# B&R Automation Studio project NAEUL004C00R13L518F00 (part 21)

#### Act_OptP0935UpdtDat.st
```iecst
ACTION Act_OptP0935UpdtDat:

	tyP0935Lifter.tyMotionStd.tyNumCurrPos.diValue			:= p_diLifterBtmActualPos;
	tyP0935Lifter.tyMotionStd.tyNumErrCode.diValue			:= UDINT_TO_DINT(p_udiLifterBtmAxisErrID);
	tyP0935Lifter.tyMotionStd.tyBitmapPwr.usiValueIdx		:= BOOL_TO_USINT(p_bLifterBtmPwrOn);
	tyP0935Lifter.tyMotionStd.tyBitmapRst.usiValueIdx		:= BOOL_TO_USINT(NOT p_bLifterBtmAxisErr);
	tyP0935Lifter.tyMotionStd.tyBitmapOrigin.usiValueIdx	:= BOOL_TO_USINT(p_bLifterBtmIsHomed);
	tyP0935Lifter.tyMotionStd.tyBtnUpLmtSen.bValue			:= p_bLifterBtmUpSen;
	tyP0935Lifter.tyMotionStd.tyBtnDownLmtSen.bValue		:= p_bLifterBtmDownSen;

	//Machine Bitmap
	IF p_bLifterBtmIsHomed = TRUE THEN
		IF p_diLifterBtmActualPos <= (p_tyNtParamCurr.tyUILifterTargetPos.diMax / 3) THEN
			tyP0935Lifter.tyMotionStd.tyBitmapMc.uiValueIdx 	:= 2;
		ELSIF p_diLifterBtmActualPos <= (p_tyNtParamCurr.tyUILifterTargetPos.diMax / 3 * 2) THEN
			tyP0935Lifter.tyMotionStd.tyBitmapMc.uiValueIdx 	:= 3;
		ELSE
			tyP0935Lifter.tyMotionStd.tyBitmapMc.uiValueIdx 	:= 4;
		END_IF
	ELSE
		tyP0935Lifter.tyMotionStd.tyBitmapMc.uiValueIdx	:= 2;
	END_IF

//	IF p_tyNtParamCurr.eProjMag = ULMagTriple THEN
//		tyP0935Lifter.tyMotionStd.tyBitmapMc.uiValueIdx	:= tyP0935Lifter.tyMotionStd.tyBitmapMc.uiValueIdx + 100;
//	END_IF

	IF p_tyNtParamCurr.eProjMag = ULMagDual THEN
		IF p_tyNtParamCurr.bProjLifterMagPlatform AND p_tyNtParamCurr.bUIConvDirRL THEN
			IF 	tyP0935Lifter.tyMotionStd.tyBitmapMc.uiValueIdx < 700 THEN
				tyP0935Lifter.tyMotionStd.tyBitmapMc.uiValueIdx	:= tyP0935Lifter.tyMotionStd.tyBitmapMc.uiValueIdx + 700;
			END_IF
		ELSIF p_tyNtParamCurr.bProjLifterMagPlatform THEN
			IF p_tyNtParamCurr.bProjMagConvLane1Prep = FALSE THEN
				IF 	tyP0935Lifter.tyMotionStd.tyBitmapMc.uiValueIdx < 600 THEN
					tyP0935Lifter.tyMotionStd.tyBitmapMc.uiValueIdx	:= tyP0935Lifter.tyMotionStd.tyBitmapMc.uiValueIdx + 600;
				END_IF
			ELSE
				IF 	tyP0935Lifter.tyMotionStd.tyBitmapMc.uiValueIdx < 900 THEN //Lifter1 - 902,903,904
					tyP0935Lifter.tyMotionStd.tyBitmapMc.uiValueIdx	:= tyP0935Lifter.tyMotionStd.tyBitmapMc.uiValueIdx + 900;
				END_IF
			END_IF
		ELSIF p_tyNtParamCurr.bMagAutoVerifyPrep = FALSE THEN
			IF 	tyP0935Lifter.tyMotionStd.tyBitmapMc.uiValueIdx < 100 THEN
				tyP0935Lifter.tyMotionStd.tyBitmapMc.uiValueIdx	:= tyP0935Lifter.tyMotionStd.tyBitmapMc.uiValueIdx + 300;
			END_IF
		ELSE
			IF 	tyP0935Lifter.tyMotionStd.tyBitmapMc.uiValueIdx < 300 THEN
				tyP0935Lifter.tyMotionStd.tyBitmapMc.uiValueIdx	:= tyP0935Lifter.tyMotionStd.tyBitmapMc.uiValueIdx + 300;
			END_IF
		END_IF
	ELSIF p_tyNtParamCurr.eProjMag = ULMagTriple THEN
		IF p_tyNtParamCurr.bProjLifterMagPlatform AND p_tyNtParamCurr.bUIConvDirRL THEN
			IF 	tyP0935Lifter.tyMotionStd.tyBitmapMc.uiValueIdx < 800 THEN
				tyP0935Lifter.tyMotionStd.tyBitmapMc.uiValueIdx	:= tyP0935Lifter.tyMotionStd.tyBitmapMc.uiValueIdx + 800;
			END_IF
		ELSIF p_tyNtParamCurr.bProjLifterMagPlatform THEN
			IF tyP0935Lifter.tyMotionStd.tyBitmapMc.uiValueIdx < 500 THEN
				tyP0935Lifter.tyMotionStd.tyBitmapMc.uiValueIdx	:= tyP0935Lifter.tyMotionStd.tyBitmapMc.uiValueIdx + 500;
			END_IF
		ELSIF p_tyNtParamCurr.bProjMotorizedPusherPrep = FALSE THEN //p_tyNtParamCurr.bMagAutoVerifyPrep = TRUE AND p_tyNtParamCurr.bProjMotorizedPusherPrep = FALSE THEN
			IF 	tyP0935Lifter.tyMotionStd.tyBitmapMc.uiValueIdx < 200 THEN
				tyP0935Lifter.tyMotionStd.tyBitmapMc.uiValueIdx	:= tyP0935Lifter.tyMotionStd.tyBitmapMc.uiValueIdx + 200;
			END_IF
		ELSIF  p_tyNtParamCurr.bMagAutoVerifyPrep = FALSE AND p_tyNtParamCurr.bProjMotorizedPusherPrep = TRUE THEN
			IF 	tyP0935Lifter.tyMotionStd.tyBitmapMc.uiValueIdx < 400 AND p_tyNtParamCurr.bCurtainSenPrep  THEN

				tyP0935Lifter.tyMotionStd.tyBitmapMc.uiValueIdx	:= tyP0935Lifter.tyMotionStd.tyBitmapMc.uiValueIdx + 440;
			ELSE
				tyP0935Lifter.tyMotionStd.tyBitmapMc.uiValueIdx	:= tyP0935Lifter.tyMotionStd.tyBitmapMc.uiValueIdx + 400;
			END_IF
		END_IF
	END_IF

END_ACTION
```

#### Act_OptP0935Keypad.st
```iecst
ACTION Act_OptP0935Keypad:

	IF fUIOutRtStatTPIsOpen(ADR(tyP0935Lifter.tyMotionStd.tyNumTargetPos.uiRtStat)) = TRUE THEN
		tyProperty.tyKeypad.tyStringTitle.sKeypadTitle	:= tyP0935Lifter.tyMotionStd.tyNumTargetPos.sKeypadTitle;

	ELSIF fUIOutRtStatTPIsOpen(ADR(tyP0935Lifter.tyMotionStd.tyNumStepSize.uiRtStat)) = TRUE THEN
		tyProperty.tyKeypad.tyStringTitle.sKeypadTitle	:= tyP0935Lifter.tyMotionStd.tyNumStepSize.sKeypadTitle;

	ELSIF fUIOutRtStatTPIsOpen(ADR(tyP0935Lifter.tyMotionStd.tyNumNomSpd.uiRtStat)) = TRUE THEN
		tyProperty.tyKeypad.tyStringTitle.sKeypadTitle	:= tyP0935Lifter.tyMotionStd.tyNumNomSpd.sKeypadTitle;

	ELSIF fUIOutRtStatTPIsOpen(ADR(tyP0935Lifter.tyMotionStd.tyNumSlwSpd.uiRtStat)) = TRUE THEN
		tyProperty.tyKeypad.tyStringTitle.sKeypadTitle	:= tyP0935Lifter.tyMotionStd.tyNumSlwSpd.sKeypadTitle;

	ELSIF fUIOutRtStatTPIsOpen(ADR(tyP0935Lifter.tyLifter.tyNumNewSlt.uiRtStat)) = TRUE THEN
		tyProperty.tyKeypad.tyStringTitle.sKeypadTitle	:= tyP0935Lifter.tyLifter.tyNumNewSlt.sKeypadTitle;

	ELSIF fUIOutRtStatTPIsOpen(ADR(tyP0935Lifter.tyLifter.tyNumMagPos.uiRtStat)) = TRUE THEN
		tyProperty.tyKeypad.tyStringTitle.sKeypadTitle	:= tyP0935Lifter.tyLifter.tyNumMagPos.sKeypadTitle;

	END_IF

END_ACTION
```

#### Act_OptP0935RstMnl.st
```iecst
ACTION Act_OptP0935RstMnl:

	IF EDGEPOS((bManualMod = FALSE) OR (p_eLifterBtmStatus = Error)) THEN

		eLifterBtmAct	:= LifterActIdle;

		bJogSlow				:= FALSE;
		bJogFast				:= FALSE;
		fbJogSlowToFastDlyTm.IN	:= FALSE;

		tyP0935Lifter.tyLifter.tyBtnGo.bRtCompl					:= FALSE;
		tyP0935Lifter.tyLifter.tyBtnNxtSlt.bRtCompl				:= FALSE;
		tyP0935Lifter.tyLifter.tyBtnPrevSlt.bRtCompl			:= FALSE;
		tyP0935Lifter.tyLifter.tyBtnGoLaneA.bRtCompl			:= FALSE;
		tyP0935Lifter.tyLifter.tyBtnGoLaneB.bRtCompl			:= FALSE;
		tyP0935Lifter.tyLifter.tyBtnGoLaneD_G.bRtCompl			:= FALSE;
		tyP0935Lifter.tyLifter.tyBtnGoLaneE_H.bRtCompl			:= FALSE;

		tyP0935Lifter.tyLifter.tyBtnGo.bValue					:= FALSE;
		tyP0935Lifter.tyLifter.tyBtnNxtSlt.bValue				:= FALSE;
		tyP0935Lifter.tyLifter.tyBtnPrevSlt.bValue				:= FALSE;
		tyP0935Lifter.tyLifter.tyBtnGoLaneA.bValue				:= FALSE;
		tyP0935Lifter.tyLifter.tyBtnGoLaneB.bValue				:= FALSE;
		tyP0935Lifter.tyLifter.tyBtnGoLaneD_G.bValue				:= FALSE;
		tyP0935Lifter.tyLifter.tyBtnGoLaneE_H.bValue				:= FALSE;

		tyP0935Lifter.tyLifter.tyBtnGo.bRtLk					:= FALSE;
		tyP0935Lifter.tyLifter.tyBtnNxtSlt.bRtLk				:= FALSE;
		tyP0935Lifter.tyLifter.tyBtnPrevSlt.bRtLk				:= FALSE;
		tyP0935Lifter.tyLifter.tyBtnGoLaneA.bRtLk				:= FALSE;
		tyP0935Lifter.tyLifter.tyBtnGoLaneB.bRtLk				:= FALSE;
		tyP0935Lifter.tyLifter.tyBtnGoLaneD_G.bRtLk				:= FALSE;
		tyP0935Lifter.tyLifter.tyBtnGoLaneE_H.bRtLk				:= FALSE;

		tyP0935Lifter.tyLifter.tyBtnGo.uiMaskRtStat.0			:= FALSE;
		tyP0935Lifter.tyLifter.tyBtnNxtSlt.uiMaskRtStat.0		:= FALSE;
		tyP0935Lifter.tyLifter.tyBtnPrevSlt.uiMaskRtStat.0		:= FALSE;
		tyP0935Lifter.tyLifter.tyBtnGoLaneA.uiMaskRtStat.0		:= FALSE;
		tyP0935Lifter.tyLifter.tyBtnGoLaneB.uiMaskRtStat.0		:= FALSE;
		tyP0935Lifter.tyLifter.tyBtnGoLaneD_G.uiMaskRtStat.0		:= FALSE;
		tyP0935Lifter.tyLifter.tyBtnGoLaneE_H.uiMaskRtStat.0		:= FALSE;

		tyP0935Lifter.tyMotionStd.tyBtnPwr.bRtCompl				:= FALSE;
		tyP0935Lifter.tyMotionStd.tyBtnStop.bRtCompl			:= FALSE;
		tyP0935Lifter.tyMotionStd.tyBtnOrigin.bRtCompl			:= FALSE;
		tyP0935Lifter.tyMotionStd.tyBtnRst.bRtCompl				:= FALSE;
		tyP0935Lifter.tyMotionStd.tyBtnMovAbs.bRtCompl			:= FALSE;
		tyP0935Lifter.tyMotionStd.tyBtnMovRel.bRtCompl			:= FALSE;
		tyP0935Lifter.tyMotionStd.tyBtnJogUp.bRtCompl			:= FALSE;
		tyP0935Lifter.tyMotionStd.tyBtnJogDown.bRtCompl			:= FALSE;

		tyP0935Lifter.tyMotionStd.tyBtnPwr.bValue				:= FALSE;
		tyP0935Lifter.tyMotionStd.tyBtnStop.bValue				:= TRUE;
		tyP0935Lifter.tyMotionStd.tyBtnOrigin.bValue			:= FALSE;
		tyP0935Lifter.tyMotionStd.tyBtnRst.bValue				:= FALSE;
		tyP0935Lifter.tyMotionStd.tyBtnMovAbs.bValue			:= FALSE;
		tyP0935Lifter.tyMotionStd.tyBtnMovRel.bValue			:= FALSE;
		tyP0935Lifter.tyMotionStd.tyBtnJogUp.bValue				:= FALSE;
		tyP0935Lifter.tyMotionStd.tyBtnJogDown.bValue			:= FALSE;

		tyP0935Lifter.tyMotionStd.tyBtnPwr.bRtLk				:= FALSE;
		tyP0935Lifter.tyMotionStd.tyBtnStop.bRtLk				:= TRUE;
		tyP0935Lifter.tyMotionStd.tyBtnOrigin.bRtLk				:= FALSE;
		tyP0935Lifter.tyMotionStd.tyBtnRst.bRtLk				:= FALSE;
		tyP0935Lifter.tyMotionStd.tyBtnMovAbs.bRtLk				:= FALSE;
		tyP0935Lifter.tyMotionStd.tyBtnMovRel.bRtLk				:= FALSE;
		tyP0935Lifter.tyMotionStd.tyBtnJogUp.bRtLk				:= FALSE;
		tyP0935Lifter.tyMotionStd.tyBtnJogDown.bRtLk			:= FALSE;

		tyP0935Lifter.tyMotionStd.tyBtnPwr.uiMaskRtStat			:= TRUE;
		tyP0935Lifter.tyMotionStd.tyBtnOrigin.uiMaskRtStat		:= FALSE;
		tyP0935Lifter.tyMotionStd.tyBtnRst.uiMaskRtStat			:= TRUE;
		tyP0935Lifter.tyMotionStd.tyBtnMovAbs.uiMaskRtStat		:= FALSE;
		tyP0935Lifter.tyMotionStd.tyBtnMovRel.uiMaskRtStat		:= FALSE;
		tyP0935Lifter.tyMotionStd.tyBtnJogUp.uiMaskRtStat		:= FALSE;
		tyP0935Lifter.tyMotionStd.tyBtnJogDown.uiMaskRtStat		:= FALSE;

	END_IF

	eInShutterAct	:= PneuActIdle;
	eOutShutterAct	:= PneuActIdle;

	tyP0935Lifter.tyInOutletShutterFB.tyBtnClose.bRtCompl	:= FALSE;
	tyP0935Lifter.tyInOutletShutterFB.tyBtnClose.bValue	:= FALSE;
	tyP0935Lifter.tyInOutletShutterFB.tyBtnOpen.bRtCompl	:= FALSE;
	tyP0935Lifter.tyInOutletShutterFB.tyBtnOpen.bValue	:= FALSE;

END_ACTION
```

#### Act_EntP0936Disp.st
```iecst
ACTION Act_EntP0936Disp:

	//Access Address
	p_tyC0001MotionStd ACCESS ADR(tyP0936Trav.tyMotionStd);

	p_tyC0002FullMask ACCESS ADR(tyP0936Trav.tyFullMaskHide);

	p_tyC0004Navi ACCESS ADR(tyP0936Trav.tyNaviBack);

	p_tyC0005Main ACCESS ADR(tyCommon.tyMain);

	p_tyC0007Notif ACCESS ADR(tyCommon.tyNotif);

	p_tyC0008MsgBox ACCESS ADR(tyP0936Trav.tyMsgBoxHide);

	p_tyC0009Info ACCESS ADR(tyCommon.tyInfo);

	p_tyP0936Trav ACCESS ADR(tyP0936Trav.tyTrav);

	p_tyP0936InOutletShutterFB ACCESS ADR(tyP0936Trav.tyInOutletShutterFB);

	//Display
	tyP0936Trav.tyMotionStd.tyBtnPwr.bValue	:= p_bTravPwrOn;

END_ACTION
```

#### Act_OptP0936Navi.st
```iecst
ACTION Act_OptP0936Navi:

	IF tyP0936Trav.tyNaviBack.tyBtnBack.bRtCompl = TRUE THEN
		eChgPage		:= UIP0920MtrNPneuCtrl;

		tyP0936Trav.tyNaviBack.tyBtnBack.bRtCompl			:= FALSE;
		tyP0936Trav.tyNaviBack.tyBtnBack.bValue				:= FALSE;

	END_IF

END_ACTION
```

#### Act_OptP0936FullMask.st
```iecst
ACTION Act_OptP0936FullMask:

	IF eCurrPage = UIP0936Trav THEN

		IF p_tyDI.bEStopSig = FALSE THEN
			p_tyC0002FullMask ACCESS ADR(tyP0936Trav.tyFullMaskEStop);

		ELSIF p_tyDI.bCoverSWSig = FALSE THEN
			p_tyC0002FullMask ACCESS ADR(tyP0936Trav.tyFullMaskCWSig);

		ELSIF p_tyDI.bSafetyRlySig = FALSE THEN
			p_tyC0002FullMask ACCESS ADR(tyP0936Trav.tyFullMaskSafetyRly);

		ELSIF p_tyDI.bConvLftSen THEN
			p_tyC0002FullMask ACCESS ADR(tyP0936Trav.tyFullMaskLftSenInterrupt);

		ELSIF p_tyDI.bConvClrSen THEN
			p_tyC0002FullMask ACCESS ADR(tyP0936Trav.tyFullMaskClrSenInterrupt);

		ELSIF p_tyDI.bPusherExtRS = TRUE THEN
			p_tyC0002FullMask ACCESS ADR(tyP0936Trav.tyFullMaskPshrInterrupt);
		ELSIF p_tyDI.bPusherRetRS = FALSE AND p_tyDI.bPusherRetSlwSen = FALSE  THEN
			p_tyC0002FullMask ACCESS ADR(tyP0936Trav.tyFullMaskPshrNotRetInterrupt);
		ELSIF (p_tyNtParamCurr.bProjInletShutPrep AND p_tyDI.bInShutterCloseRS = FALSE) AND NOT(bBypassShutForCalib) THEN
			p_tyC0002FullMask ACCESS ADR(tyP0936Trav.tyFullMaskInShutOpnInterrupt);

		ELSIF  ((p_tyDI.bOutShutterCloseRS = FALSE AND p_tyNtParamCurr.bProjOutletShutPrep) OR (p_tyDI.bOutShutterCloseRS2 = FALSE AND p_tyNtParamCurr.bProjOutletShut2Prep )OR (p_tyDI.bOutShutterCloseRS3 = FALSE AND p_tyNtParamCurr.bProjOutletShut3Prep)) AND NOT(bBypassShutForCalib) THEN
			IF p_tyNtParamCurr.bCurtainSenPrep THEN
				IF (p_tyDI.bOutShutterCloseRS = FALSE AND p_tyNtParamCurr.bProjOutletShutPrep) OR (p_tyDI.bOutShutterCloseRS2 = FALSE AND p_tyNtParamCurr.bProjOutletShut2Prep)OR (p_tyDI.bOutShutterCloseRS3 = FALSE AND p_tyNtParamCurr.bProjOutletShut3Prep )THEN
					p_tyC0002FullMask ACCESS ADR(tyP0936Trav.tyFullMaskOutShutOpnInterrupt);
				END_IF
			ELSE
				IF p_tyDI.bOutShutterCloseRS = FALSE THEN
					p_tyC0002FullMask ACCESS ADR(tyP0936Trav.tyFullMaskOutShutOpnInterrupt);
				END_IF
			END_IF
		ELSE
			p_tyC0002FullMask ACCESS ADR(tyP0936Trav.tyFullMaskHide);

		END_IF

	END_IF

END_ACTION
```

#### Act_OptP0936FBCtrl.st
```iecst
ACTION Act_OptP0936FBCtrl:

	fbJogSlowToFastDlyTm.PT			:= T#2s;
	fbJogSlowToFastDlyTm;
	fbLmtRstTm;

//	IF EDGEPOS((p_udiTravAxisErrID = 21570 OR p_udiTravAxisErrID = 21571)
	IF EDGEPOS ((p_bTravFwdLmtSen OR p_bTravRevLmtSen OR p_udiTravAxisErrID = 21570 OR p_udiTravAxisErrID = 21571)
		AND tyP0936Trav.tyMotionStd.tyBtnJogRear.bValue = FALSE
		AND tyP0936Trav.tyMotionStd.tyBtnJogFront.bValue = FALSE)
	THEN
		fbLmtRstTm.IN				:= TRUE;
	END_IF

	IF fbLmtRstTm.Q = TRUE THEN
		tyP0936Trav.tyMotionStd.tyBtnRst.bRtCompl		:= TRUE;
	END_IF

	IF (tyP0936Trav.tyMotionStd.tyBtnJogFront.bValue = FALSE AND tyP0936Trav.tyMotionStd.tyBtnJogRear.bValue = FALSE) AND (p_bTravJogging = TRUE) THEN
		bJogStopTrav	:= TRUE;
	END_IF

	IF tyP0936Trav.tyMotionStd.tyBtnStop.bRtCompl = TRUE THEN
		eTravAct		:= TravActStop;

		IF p_eTravStat = TravActStop AND p_eTravStatus = Done THEN
			eTravAct	:= TravActIdle;

			tyP0936Trav.tyMotionStd.tyBtnStop.bRtCompl			:= FALSE;
			tyP0936Trav.tyMotionStd.tyBtnJogRear.bRtCompl		:= FALSE;
			tyP0936Trav.tyMotionStd.tyBtnJogFront.bRtCompl		:= FALSE;
			tyP0936Trav.tyMotionStd.tyBtnOrigin.bRtCompl		:= FALSE;
			tyP0936Trav.tyMotionStd.tyBtnMovAbs.bRtCompl		:= FALSE;
			tyP0936Trav.tyMotionStd.tyBtnMovRel.bRtCompl		:= FALSE;
			tyP0936Trav.tyTrav.tyBtnGoToLaneA.bRtCompl			:= FALSE;
			tyP0936Trav.tyTrav.tyBtnGoToLaneB.bRtCompl			:= FALSE;
			tyP0936Trav.tyTrav.tyBtnGoToMag1.bRtCompl			:= FALSE;
			tyP0936Trav.tyTrav.tyBtnGoToMag2.bRtCompl			:= FALSE;
			tyP0936Trav.tyTrav.tyBtnGoToMag3.bRtCompl			:= FALSE;

			tyP0936Trav.tyMotionStd.tyBtnStop.bValue			:= TRUE;
			tyP0936Trav.tyMotionStd.tyBtnJogRear.bValue			:= FALSE;
			tyP0936Trav.tyMotionStd.tyBtnJogFront.bValue		:= FALSE;
			tyP0936Trav.tyMotionStd.tyBtnOrigin.bValue			:= FALSE;
			tyP0936Trav.tyMotionStd.tyBtnMovAbs.bValue			:= FALSE;
			tyP0936Trav.tyMotionStd.tyBtnMovRel.bValue			:= FALSE;
			tyP0936Trav.tyTrav.tyBtnGoToLaneA.bValue			:= FALSE;
			tyP0936Trav.tyTrav.tyBtnGoToLaneB.bValue			:= FALSE;
			tyP0936Trav.tyTrav.tyBtnGoToMag1.bValue				:= FALSE;
			tyP0936Trav.tyTrav.tyBtnGoToMag2.bValue				:= FALSE;
			tyP0936Trav.tyTrav.tyBtnGoToMag3.bValue				:= FALSE;

			tyP0936Trav.tyMotionStd.tyBtnStop.bRtLk				:= TRUE;
			tyP0936Trav.tyMotionStd.tyBtnJogRear.bRtLk			:= FALSE;
			tyP0936Trav.tyMotionStd.tyBtnJogFront.bRtLk			:= FALSE;
			tyP0936Trav.tyMotionStd.tyBtnOrigin.bRtLk			:= FALSE;
			tyP0936Trav.tyMotionStd.tyBtnMovAbs.bRtLk			:= FALSE;
			tyP0936Trav.tyMotionStd.tyBtnMovRel.bRtLk			:= FALSE;
			tyP0936Trav.tyTrav.tyBtnGoToLaneA.bRtLk				:= FALSE;
			tyP0936Trav.tyTrav.tyBtnGoToLaneB.bRtLk				:= FALSE;
			tyP0936Trav.tyTrav.tyBtnGoToMag1.bRtLk				:= FALSE;
			tyP0936Trav.tyTrav.tyBtnGoToMag2.bRtLk				:= FALSE;
			tyP0936Trav.tyTrav.tyBtnGoToMag3.bRtLk				:= FALSE;
		END_IF

	ELSIF (tyP0936Trav.tyMotionStd.tyBtnJogRear.bRtCompl = TRUE) OR (tyP0936Trav.tyMotionStd.tyBtnJogFront.bRtCompl = TRUE) OR (bJogStopTrav = TRUE) THEN
		bJogSlow					:= FALSE;
		bJogFast					:= FALSE;

		fbJogSlowToFastDlyTm.IN		:= FALSE;

		eTravAct		:= TravActJogStop;

		IF p_eTravStat = TravActJogStop AND p_eTravStatus = Done THEN
			eTravAct		:= TravActIdle;

			bJogStopTrav	:= FALSE;

			tyP0936Trav.tyMotionStd.tyBtnStop.bRtCompl			:= FALSE;
			tyP0936Trav.tyMotionStd.tyBtnJogRear.bRtCompl		:= FALSE;
			tyP0936Trav.tyMotionStd.tyBtnJogFront.bRtCompl		:= FALSE;
			tyP0936Trav.tyMotionStd.tyBtnOrigin.bRtCompl		:= FALSE;
			tyP0936Trav.tyMotionStd.tyBtnMovAbs.bRtCompl		:= FALSE;
			tyP0936Trav.tyMotionStd.tyBtnMovRel.bRtCompl		:= FALSE;
			tyP0936Trav.tyTrav.tyBtnGoToLaneA.bRtCompl			:= FALSE;
			tyP0936Trav.tyTrav.tyBtnGoToLaneB.bRtCompl			:= FALSE;
			tyP0936Trav.tyTrav.tyBtnGoToMag1.bRtCompl			:= FALSE;
			tyP0936Trav.tyTrav.tyBtnGoToMag2.bRtCompl			:= FALSE;
			tyP0936Trav.tyTrav.tyBtnGoToMag3.bRtCompl			:= FALSE;

			tyP0936Trav.tyMotionStd.tyBtnStop.bValue			:= TRUE;
			tyP0936Trav.tyMotionStd.tyBtnJogRear.bValue			:= FALSE;
			tyP0936Trav.tyMotionStd.tyBtnJogFront.bValue		:= FALSE;
			tyP0936Trav.tyMotionStd.tyBtnOrigin.bValue			:= FALSE;
			tyP0936Trav.tyMotionStd.tyBtnMovAbs.bValue			:= FALSE;
			tyP0936Trav.tyMotionStd.tyBtnMovRel.bValue			:= FALSE;
			tyP0936Trav.tyTrav.tyBtnGoToLaneA.bValue			:= FALSE;
			tyP0936Trav.tyTrav.tyBtnGoToLaneB.bValue			:= FALSE;
			tyP0936Trav.tyTrav.tyBtnGoToMag1.bValue				:= FALSE;
			tyP0936Trav.tyTrav.tyBtnGoToMag2.bValue				:= FALSE;
			tyP0936Trav.tyTrav.tyBtnGoToMag3.bValue				:= FALSE;

			tyP0936Trav.tyMotionStd.tyBtnStop.bRtLk				:= TRUE;
			tyP0936Trav.tyMotionStd.tyBtnJogRear.bRtLk			:= FALSE;
			tyP0936Trav.tyMotionStd.tyBtnJogFront.bRtLk			:= FALSE;
			tyP0936Trav.tyMotionStd.tyBtnOrigin.bRtLk			:= FALSE;
			tyP0936Trav.tyMotionStd.tyBtnMovAbs.bRtLk			:= FALSE;
			tyP0936Trav.tyMotionStd.tyBtnMovRel.bRtLk			:= FALSE;
			tyP0936Trav.tyTrav.tyBtnGoToLaneA.bRtLk				:= FALSE;
			tyP0936Trav.tyTrav.tyBtnGoToLaneB.bRtLk				:= FALSE;
			tyP0936Trav.tyTrav.tyBtnGoToMag1.bRtLk				:= FALSE;
			tyP0936Trav.tyTrav.tyBtnGoToMag2.bRtLk				:= FALSE;
			tyP0936Trav.tyTrav.tyBtnGoToMag3.bRtLk				:= FALSE;

		END_IF

	ELSIF tyP0936Trav.tyMotionStd.tyBtnPwr.bRtCompl = TRUE THEN
		tyP0936Trav.tyMotionStd.tyBtnPwr.bRtLk					:= TRUE;

		IF tyP0936Trav.tyMotionStd.tyBtnPwr.bValue = TRUE THEN
			eTravAct		:= TravActPwrOn;

			IF p_eTravStat = TravActPwrOn AND p_eTravStatus = Done THEN
				eTravAct	:= TravActIdle;

				tyP0936Trav.tyMotionStd.tyBtnPwr.bRtCompl		:= FALSE;
				tyP0936Trav.tyMotionStd.tyBtnPwr.bRtLk			:= FALSE;
			END_IF
		ELSE
			eTravAct		:= TravActPwrOff;

			IF p_eTravStat = TravActPwrOff AND p_eTravStatus = Done THEN
				eTravAct	:= TravActIdle;

				tyP0936Trav.tyMotionStd.tyBtnPwr.bRtCompl		:= FALSE;
				tyP0936Trav.tyMotionStd.tyBtnPwr.bRtLk			:= FALSE;
			END_IF
		END_IF

	ELSIF tyP0936Trav.tyMotionStd.tyBtnOrigin.bRtCompl = TRUE THEN
		tyP0936Trav.tyMotionStd.tyBtnOrigin.bValue				:= TRUE;
		tyP0936Trav.tyMotionStd.tyBtnStop.bValue				:= FALSE;

		tyP0936Trav.tyMotionStd.tyBtnOrigin.bRtLk				:= TRUE;
		tyP0936Trav.tyMotionStd.tyBtnStop.bRtLk					:= FALSE;

		eTravAct		:= TravActHoming;

		IF p_eTravStat = TravActHoming AND p_eTravStatus = Done THEN
			eTravAct	:= TravActIdle;

			tyP0936Trav.tyMotionStd.tyBtnOrigin.bRtCompl		:= FALSE;
			tyP0936Trav.tyMotionStd.tyBtnOrigin.bValue			:= FALSE;
			tyP0936Trav.tyMotionStd.tyBtnStop.bValue			:= TRUE;

			tyP0936Trav.tyMotionStd.tyBtnOrigin.bRtLk			:= FALSE;
			tyP0936Trav.tyMotionStd.tyBtnStop.bRtLk				:= TRUE;
		END_IF

	ELSIF tyP0936Trav.tyMotionStd.tyBtnRst.bRtCompl = TRUE THEN
		tyP0936Trav.tyMotionStd.tyBtnRst.bValue					:= TRUE;
		tyP0936Trav.tyMotionStd.tyBtnRst.bRtLk					:= TRUE;

		eTravAct		:= TravActRstAxisErr;

		IF p_eTravStat = TravActRstAxisErr AND p_eTravStatus = Done THEN
			eTravAct	:= TravActIdle;

			tyP0936Trav.tyMotionStd.tyBtnRst.bRtCompl			:= FALSE;
			tyP0936Trav.tyMotionStd.tyBtnRst.bValue				:= FALSE;
			tyP0936Trav.tyMotionStd.tyBtnRst.bRtLk				:= FALSE;

			fbLmtRstTm.IN			:= FALSE;
		END_IF

	ELSIF tyP0936Trav.tyTrav.tyBtnGoToLaneA.bRtCompl = TRUE THEN
		tyP0936Trav.tyTrav.tyBtnGoToLaneA.bValue				:= TRUE;
		tyP0936Trav.tyMotionStd.tyBtnStop.bValue				:= FALSE;

		tyP0936Trav.tyTrav.tyBtnGoToLaneA.bRtLk					:= TRUE;
		tyP0936Trav.tyMotionStd.tyBtnStop.bRtLk					:= FALSE;

		diMnlTravNomSpd	:= tyP0936Trav.tyMotionStd.tyNumNomSpd.diValue;

		eTravAct		:= TravActGoAPos;

		IF p_eTravStat = TravActGoAPos AND p_eTravStatus = Done THEN
			eTravAct	:= TravActIdle;

			tyP0936Trav.tyTrav.tyBtnGoToLaneA.bRtCompl				:= FALSE;
			tyP0936Trav.tyTrav.tyBtnGoToLaneA.bValue				:= FALSE;
			tyP0936Trav.tyMotionStd.tyBtnStop.bValue				:= TRUE;

			tyP0936Trav.tyTrav.tyBtnGoToLaneA.bRtLk					:= FALSE;
			tyP0936Trav.tyMotionStd.tyBtnStop.bRtLk					:= TRUE;
		END_IF

	ELSIF tyP0936Trav.tyTrav.tyBtnGoToLaneB.bRtCompl = TRUE THEN
		tyP0936Trav.tyTrav.tyBtnGoToLaneB.bValue					:= TRUE;
		tyP0936Trav.tyMotionStd.tyBtnStop.bValue					:= FALSE;

		tyP0936Trav.tyTrav.tyBtnGoToLaneB.bRtLk						:= TRUE;
		tyP0936Trav.tyMotionStd.tyBtnStop.bRtLk						:= FALSE;

		diMnlTravNomSpd	:= tyP0936Trav.tyMotionStd.tyNumNomSpd.diValue;

		eTravAct		:= TravActGoBPos;

		IF p_eTravStat = TravActGoBPos AND p_eTravStatus = Done THEN
			eTravAct	:= TravActIdle;

			tyP0936Trav.tyTrav.tyBtnGoToLaneB.bRtCompl				:= FALSE;
			tyP0936Trav.tyTrav.tyBtnGoToLaneB.bValue				:= FALSE;
			tyP0936Trav.tyMotionStd.tyBtnStop.bValue				:= TRUE;

			tyP0936Trav.tyTrav.tyBtnGoToLaneB.bRtLk					:= FALSE;
			tyP0936Trav.tyMotionStd.tyBtnStop.bRtLk					:= TRUE;
		END_IF

	ELSIF tyP0936Trav.tyTrav.tyBtnGoToMag1.bRtCompl = TRUE THEN
		tyP0936Trav.tyTrav.tyBtnGoToMag1.bValue						:= TRUE;
		tyP0936Trav.tyMotionStd.tyBtnStop.bValue					:= FALSE;

		tyP0936Trav.tyTrav.tyBtnGoToMag1.bRtLk						:= TRUE;
		tyP0936Trav.tyMotionStd.tyBtnStop.bRtLk						:= FALSE;

		diMnlTravNomSpd	:= tyP0936Trav.tyMotionStd.tyNumNomSpd.diValue;

		eTravAct		:= TravActGoDPos;

		IF p_eTravStat = TravActGoDPos AND p_eTravStatus = Done THEN
			eTravAct	:= TravActIdle;

			tyP0936Trav.tyTrav.tyBtnGoToMag1.bRtCompl				:= FALSE;
			tyP0936Trav.tyTrav.tyBtnGoToMag1.bValue					:= FALSE;
			tyP0936Trav.tyMotionStd.tyBtnStop.bValue				:= TRUE;

			tyP0936Trav.tyTrav.tyBtnGoToMag1.bRtLk					:= FALSE;
			tyP0936Trav.tyMotionStd.tyBtnStop.bRtLk					:= TRUE;
		END_IF

	ELSIF tyP0936Trav.tyTrav.tyBtnGoToMag2.bRtCompl = TRUE THEN
		tyP0936Trav.tyTrav.tyBtnGoToMag2.bValue						:= TRUE;
		tyP0936Trav.tyMotionStd.tyBtnStop.bValue					:= FALSE;

		tyP0936Trav.tyTrav.tyBtnGoToMag2.bRtLk						:= TRUE;
		tyP0936Trav.tyMotionStd.tyBtnStop.bRtLk						:= FALSE;

		diMnlTravNomSpd	:= tyP0936Trav.tyMotionStd.tyNumNomSpd.diValue;

		eTravAct		:= TravActGoEPos;

		IF p_eTravStat = TravActGoEPos AND p_eTravStatus = Done THEN
			eTravAct	:= TravActIdle;

			tyP0936Trav.tyTrav.tyBtnGoToMag2.bRtCompl				:= FALSE;
			tyP0936Trav.tyTrav.tyBtnGoToMag2.bValue					:= FALSE;
			tyP0936Trav.tyMotionStd.tyBtnStop.bValue				:= TRUE;

			tyP0936Trav.tyTrav.tyBtnGoToMag2.bRtLk					:= FALSE;
			tyP0936Trav.tyMotionStd.tyBtnStop.bRtLk					:= TRUE;
		END_IF

	ELSIF tyP0936Trav.tyTrav.tyBtnGoToMag3.bRtCompl = TRUE THEN
		tyP0936Trav.tyTrav.tyBtnGoToMag3.bValue						:= TRUE;
		tyP0936Trav.tyMotionStd.tyBtnStop.bValue					:= FALSE;

		tyP0936Trav.tyTrav.tyBtnGoToMag3.bRtLk						:= TRUE;
		tyP0936Trav.tyMotionStd.tyBtnStop.bRtLk						:= FALSE;

		diMnlTravNomSpd	:= tyP0936Trav.tyMotionStd.tyNumNomSpd.diValue;

		eTravAct		:= TravActGoFPos;

		IF p_eTravStat = TravActGoFPos AND p_eTravStatus = Done THEN
			eTravAct	:= TravActIdle;

			tyP0936Trav.tyTrav.tyBtnGoToMag3.bRtCompl				:= FALSE;
			tyP0936Trav.tyTrav.tyBtnGoToMag3.bValue					:= FALSE;
			tyP0936Trav.tyMotionStd.tyBtnStop.bValue				:= TRUE;

			tyP0936Trav.tyTrav.tyBtnGoToMag3.bRtLk					:= FALSE;
			tyP0936Trav.tyMotionStd.tyBtnStop.bRtLk					:= TRUE;
		END_IF

	ELSIF tyP0936Trav.tyMotionStd.tyBtnMovAbs.bRtCompl = TRUE THEN
		tyP0936Trav.tyMotionStd.tyBtnMovAbs.bValue				:= TRUE;
		tyP0936Trav.tyMotionStd.tyBtnStop.bValue				:= FALSE;

		tyP0936Trav.tyMotionStd.tyBtnMovAbs.bRtLk				:= TRUE;
		tyP0936Trav.tyMotionStd.tyBtnStop.bRtLk					:= FALSE;

		diMnlTravTargetPos	:= tyP0936Trav.tyMotionStd.tyNumTargetPos.diValue;
		diMnlTravNomSpd		:= tyP0936Trav.tyMotionStd.tyNumNomSpd.diValue;

		eTravAct		:= TravActMovAbs;

		IF p_eTravStat = TravActMovAbs AND p_eTravStatus = Done THEN
			eTravAct	:= TravActIdle;

			tyP0936Trav.tyMotionStd.tyBtnMovAbs.bRtCompl		:= FALSE;
			tyP0936Trav.tyMotionStd.tyBtnMovAbs.bValue			:= FALSE;
			tyP0936Trav.tyMotionStd.tyBtnStop.bValue			:= TRUE;

			tyP0936Trav.tyMotionStd.tyBtnMovAbs.bRtLk			:= FALSE;
			tyP0936Trav.tyMotionStd.tyBtnStop.bRtLk				:= TRUE;
		END_IF

	ELSIF tyP0936Trav.tyMotionStd.tyBtnMovRel.bRtCompl = TRUE THEN
		tyP0936Trav.tyMotionStd.tyBtnMovRel.bValue				:= TRUE;
		tyP0936Trav.tyMotionStd.tyBtnStop.bValue				:= FALSE;

		tyP0936Trav.tyMotionStd.tyBtnMovRel.bRtLk				:= TRUE;
		tyP0936Trav.tyMotionStd.tyBtnStop.bRtLk					:= FALSE;

		diMnlTravStepSize	:= tyP0936Trav.tyMotionStd.tyNumStepSize.diValue;
		diMnlTravNomSpd		:= tyP0936Trav.tyMotionStd.tyNumNomSpd.diValue;

		eTravAct		:= TravActMovRel;

		IF p_eTravStat = TravActMovRel AND p_eTravStatus = Done THEN
			eTravAct	:= TravActIdle;

			tyP0936Trav.tyMotionStd.tyBtnMovRel.bRtCompl		:= FALSE;
			tyP0936Trav.tyMotionStd.tyBtnMovRel.bValue			:= FALSE;
			tyP0936Trav.tyMotionStd.tyBtnStop.bValue			:= TRUE;

			tyP0936Trav.tyMotionStd.tyBtnMovRel.bRtLk			:= FALSE;
			tyP0936Trav.tyMotionStd.tyBtnStop.bRtLk				:= TRUE;
		END_IF

	ELSIF (tyP0936Trav.tyMotionStd.tyBtnJogRear.bValue = TRUE) AND (fbJogSlowToFastDlyTm.Q = FALSE) AND (bJogSlow = FALSE) THEN
		tyP0936Trav.tyMotionStd.tyBtnStop.bValue				:= FALSE;
		tyP0936Trav.tyMotionStd.tyBtnStop.bRtLk					:= FALSE;

		fbJogSlowToFastDlyTm.IN		:= TRUE;

		diMnlTravJogSpd	:= tyP0936Trav.tyMotionStd.tyNumSlwSpd.diValue;

		eTravAct		:= TravActJogRear;

		IF p_eTravStat = TravActJogRear AND p_eTravStatus = Done THEN
			eTravAct	:= TravActIdle;
			bJogSlow				:= TRUE;
		ELSIF p_eTravStatus = Error THEN
			fbJogSlowToFastDlyTm.IN	:= FALSE;
			bJogSlow				:= TRUE;
		END_IF

	ELSIF (tyP0936Trav.tyMotionStd.tyBtnJogRear.bValue = TRUE) AND (fbJogSlowToFastDlyTm.Q = TRUE) AND (bJogFast = FALSE) THEN
		tyP0936Trav.tyMotionStd.tyBtnStop.bValue					:= FALSE;
		tyP0936Trav.tyMotionStd.tyBtnStop.bRtLk						:= FALSE;

		fbJogSlowToFastDlyTm.IN		:= TRUE;

		diMnlTravJogSpd	:= tyP0936Trav.tyMotionStd.tyNumNomSpd.diValue;

		eTravAct		:= TravActJogRear;

		IF p_eTravStat = TravActJogRear AND p_eTravStatus = Done THEN
			eTravAct	:= TravActIdle;
			bJogFast				:= TRUE;
		ELSIF p_eTravStatus = Error THEN
			fbJogSlowToFastDlyTm.IN	:= FALSE;
			bJogFast				:= TRUE;
		END_IF

	ELSIF (tyP0936Trav.tyMotionStd.tyBtnJogFront.bValue = TRUE) AND (fbJogSlowToFastDlyTm.Q = FALSE) AND (bJogSlow = FALSE) THEN
		tyP0936Trav.tyMotionStd.tyBtnStop.bValue				:= FALSE;
		tyP0936Trav.tyMotionStd.tyBtnStop.bRtLk					:= FALSE;

		fbJogSlowToFastDlyTm.IN		:= TRUE;

		diMnlTravJogSpd	:= tyP0936Trav.tyMotionStd.tyNumSlwSpd.diValue;

		eTravAct		:= TravActJogFront;

		IF p_eTravStat = TravActJogFront AND p_eTravStatus = Done THEN
			eTravAct	:= TravActIdle;
			bJogSlow				:= TRUE;
		ELSIF p_eTravStatus = Error THEN
			fbJogSlowToFastDlyTm.IN	:= FALSE;
			bJogSlow				:= TRUE;
		END_IF

	ELSIF (tyP0936Trav.tyMotionStd.tyBtnJogFront.bValue = TRUE) AND (fbJogSlowToFastDlyTm.Q = TRUE) AND (bJogFast = FALSE) THEN

		tyP0936Trav.tyMotionStd.tyBtnStop.bValue				:= FALSE;
		tyP0936Trav.tyMotionStd.tyBtnStop.bRtLk					:= FALSE;

		fbJogSlowToFastDlyTm.IN		:= TRUE;

		diMnlTravJogSpd	:= tyP0936Trav.tyMotionStd.tyNumNomSpd.diValue;

		eTravAct		:= TravActJogFront;

		IF p_eTravStat = TravActJogFront AND p_eTravStatus = Done THEN
			eTravAct	:= TravActIdle;
			bJogFast	:= TRUE;
		ELSIF p_eTravStatus = Error THEN
			fbJogSlowToFastDlyTm.IN	:= FALSE;
			bJogFast				:= TRUE;
		END_IF
	END_IF

	//Shutter Control
	IF tyP0936Trav.tyInOutletShutterFB.tyBtnOpen.bRtCompl = TRUE THEN
		tyP0936Trav.tyInOutletShutterFB.tyBtnOpen.bRtCompl	:= FALSE;

		tyP0936Trav.tyInOutletShutterFB.tyBtnOpen.bValue	:= TRUE;
		tyP0936Trav.tyInOutletShutterFB.tyBtnClose.bValue	:= FALSE;

	ELSIF tyP0936Trav.tyInOutletShutterFB.tyBtnClose.bRtCompl = TRUE THEN
		tyP0936Trav.tyInOutletShutterFB.tyBtnClose.bRtCompl	:= FALSE;

		tyP0936Trav.tyInOutletShutterFB.tyBtnClose.bValue	:= TRUE;
		tyP0936Trav.tyInOutletShutterFB.tyBtnOpen.bValue	:= FALSE;
	END_IF

	IF tyP0936Trav.tyInOutletShutterFB.tyBtnOpen.bValue = TRUE THEN
		eInShutterAct	:= PneuActRet;
		eOutShutterAct	:= PneuActRet;

		IF (p_eInShutterStat = PneuActRet AND p_eInShutterStatus = Done)
			AND (p_eOutShutterStat = PneuActRet AND p_eOutShutterStatus = Done)
			THEN
			eInShutterAct	:= PneuActIdle;
			eOutShutterAct	:= PneuActIdle;
			tyP0936Trav.tyInOutletShutterFB.tyBtnOpen.bValue	:= FALSE;
		ELSIF p_eInShutterStatus = Error OR p_eOutShutterStatus = Error THEN
			tyP0936Trav.tyInOutletShutterFB.tyBtnOpen.bValue	:= FALSE;
		END_IF

	ELSIF tyP0936Trav.tyInOutletShutterFB.tyBtnClose.bValue = TRUE THEN
		eInShutterAct	:= PneuActExt;
		eOutShutterAct	:= PneuActExt;
		IF (p_eInShutterStat = PneuActExt AND p_eInShutterStatus = Done)
			AND (p_eOutShutterStat = PneuActExt AND p_eOutShutterStatus = Done)
			THEN
			eInShutterAct	:= PneuActIdle;
			eOutShutterAct	:= PneuActIdle;
			tyP0936Trav.tyInOutletShutterFB.tyBtnClose.bValue := FALSE;
		ELSIF p_eInShutterStatus = Error OR p_eOutShutterStatus = Error THEN
			tyP0936Trav.tyInOutletShutterFB.tyBtnClose.bValue := FALSE;
		END_IF
	END_IF

END_ACTION
```

#### Act_OptP0936FBStat.st
```iecst
ACTION Act_OptP0936FBStat:

	IF p_bTravAxisErr = TRUE THEN
		tyP0936Trav.tyMotionStd.tyStringStat.sValue		:= p_sTravAxisErrTxt;
	ELSE
		IF NOT(p_bTravJogging AND p_eTravStat = TravActIdle) THEN
			tyP0936Trav.tyMotionStd.tyStringStat.sValue		:= p_sTravStatTxt;
		END_IF
	END_IF

END_ACTION
```

#### Act_OptP0936Mask.st
```iecst
ACTION Act_OptP0936Mask:

	// Interlock Power
	IF p_bTravAxisErr = TRUE AND p_bTravPwrOn = FALSE THEN
		fUIInRtStatOff(ADR(tyP0936Trav.tyMotionStd.tyBtnPwr.uiMaskRtStat));
		tyP0936Trav.tyMotionStd.tyBtnPwr.bValue		:= FALSE;
	ELSE
		fUIInRtStatHide(ADR(tyP0936Trav.tyMotionStd.tyBtnPwr.uiMaskRtStat));
	END_IF

	// Interlock Others Move
	IF p_bTravAxisErr = TRUE OR p_bTravPwrOn = FALSE THEN
		fUIInRtStatOff(ADR(tyP0936Trav.tyMotionStd.tyBtnOrigin.uiMaskRtStat));
		fUIInRtStatOff(ADR(tyP0936Trav.tyMotionStd.tyBtnMovRel.uiMaskRtStat));
		fUIInRtStatOff(ADR(tyP0936Trav.tyMotionStd.tyBtnJogFront.uiMaskRtStat));
		fUIInRtStatOff(ADR(tyP0936Trav.tyMotionStd.tyBtnJogRear.uiMaskRtStat));
	ELSE
		fUIInRtStatHide(ADR(tyP0936Trav.tyMotionStd.tyBtnOrigin.uiMaskRtStat));
		fUIInRtStatHide(ADR(tyP0936Trav.tyMotionStd.tyBtnMovRel.uiMaskRtStat));
		fUIInRtStatHide(ADR(tyP0936Trav.tyMotionStd.tyBtnJogFront.uiMaskRtStat));
		fUIInRtStatHide(ADR(tyP0936Trav.tyMotionStd.tyBtnJogRear.uiMaskRtStat));
	END_IF

	// Interlock Move Absolute
	IF p_bTravAxisErr = TRUE OR p_bTravPwrOn = FALSE OR p_bTravIsHomed = FALSE THEN
		fUIInRtStatOff(ADR(tyP0936Trav.tyTrav.tyBtnGoToLaneA.uiMaskRtStat));
		fUIInRtStatOff(ADR(tyP0936Trav.tyTrav.tyBtnGoToLaneB.uiMaskRtStat));
		fUIInRtStatOff(ADR(tyP0936Trav.tyTrav.tyBtnGoToMag1.uiMaskRtStat));
		fUIInRtStatOff(ADR(tyP0936Trav.tyTrav.tyBtnGoToMag2.uiMaskRtStat));
		fUIInRtStatOff(ADR(tyP0936Trav.tyTrav.tyBtnGoToMag3.uiMaskRtStat));
		fUIInRtStatOff(ADR(tyP0936Trav.tyMotionStd.tyBtnMovAbs.uiMaskRtStat));
	ELSE
		fUIInRtStatHide(ADR(tyP0936Trav.tyTrav.tyBtnGoToLaneA.uiMaskRtStat));
		fUIInRtStatHide(ADR(tyP0936Trav.tyTrav.tyBtnGoToLaneB.uiMaskRtStat));
		fUIInRtStatHide(ADR(tyP0936Trav.tyTrav.tyBtnGoToMag1.uiMaskRtStat));
		fUIInRtStatHide(ADR(tyP0936Trav.tyTrav.tyBtnGoToMag2.uiMaskRtStat));
		fUIInRtStatHide(ADR(tyP0936Trav.tyTrav.tyBtnGoToMag3.uiMaskRtStat));
		fUIInRtStatHide(ADR(tyP0936Trav.tyMotionStd.tyBtnMovAbs.uiMaskRtStat));
	END_IF

	//Interlock Limit Sensor
	IF tyP0936Trav.tyMotionStd.tyBtnRearLmtSen.bValue = TRUE THEN
		fUIInRtStatOff(ADR(tyP0936Trav.tyMotionStd.tyBtnJogRear.uiMaskRtStat));
	END_IF

	IF tyP0936Trav.tyMotionStd.tyBtnFrontLmtSen.bValue = TRUE THEN
		fUIInRtStatOff(ADR(tyP0936Trav.tyMotionStd.tyBtnJogFront.uiMaskRtStat));
	END_IF

	// Interlock When Moving
	IF tyP0936Trav.tyMotionStd.tyBtnOrigin.bRtCompl = TRUE THEN
		fUIInRtStatOff(ADR(tyP0936Trav.tyMotionStd.tyBtnMovAbs.uiMaskRtStat));
		fUIInRtStatOff(ADR(tyP0936Trav.tyMotionStd.tyBtnMovRel.uiMaskRtStat));
		fUIInRtStatOff(ADR(tyP0936Trav.tyMotionStd.tyBtnJogFront.uiMaskRtStat));
		fUIInRtStatOff(ADR(tyP0936Trav.tyMotionStd.tyBtnJogRear.uiMaskRtStat));
		fUIInRtStatOff(ADR(tyP0936Trav.tyTrav.tyBtnGoToLaneA.uiMaskRtStat));
		fUIInRtStatOff(ADR(tyP0936Trav.tyTrav.tyBtnGoToLaneB.uiMaskRtStat));
		fUIInRtStatOff(ADR(tyP0936Trav.tyTrav.tyBtnGoToMag1.uiMaskRtStat));
		fUIInRtStatOff(ADR(tyP0936Trav.tyTrav.tyBtnGoToMag2.uiMaskRtStat));
		fUIInRtStatOff(ADR(tyP0936Trav.tyTrav.tyBtnGoToMag3.uiMaskRtStat));

	ELSIF tyP0936Trav.tyMotionStd.tyBtnMovAbs.bRtCompl = TRUE THEN
		fUIInRtStatOff(ADR(tyP0936Trav.tyMotionStd.tyBtnOrigin.uiMaskRtStat));
		fUIInRtStatOff(ADR(tyP0936Trav.tyMotionStd.tyBtnMovRel.uiMaskRtStat));
		fUIInRtStatOff(ADR(tyP0936Trav.tyMotionStd.tyBtnJogFront.uiMaskRtStat));
		fUIInRtStatOff(ADR(tyP0936Trav.tyMotionStd.tyBtnJogRear.uiMaskRtStat));
		fUIInRtStatOff(ADR(tyP0936Trav.tyTrav.tyBtnGoToLaneA.uiMaskRtStat));
		fUIInRtStatOff(ADR(tyP0936Trav.tyTrav.tyBtnGoToLaneB.uiMaskRtStat));
		fUIInRtStatOff(ADR(tyP0936Trav.tyTrav.tyBtnGoToMag1.uiMaskRtStat));
		fUIInRtStatOff(ADR(tyP0936Trav.tyTrav.tyBtnGoToMag2.uiMaskRtStat));
		fUIInRtStatOff(ADR(tyP0936Trav.tyTrav.tyBtnGoToMag3.uiMaskRtStat));

	ELSIF tyP0936Trav.tyMotionStd.tyBtnMovRel.bRtCompl = TRUE THEN
		fUIInRtStatOff(ADR(tyP0936Trav.tyMotionStd.tyBtnOrigin.uiMaskRtStat));
		fUIInRtStatOff(ADR(tyP0936Trav.tyMotionStd.tyBtnMovAbs.uiMaskRtStat));
		fUIInRtStatOff(ADR(tyP0936Trav.tyMotionStd.tyBtnJogFront.uiMaskRtStat));
		fUIInRtStatOff(ADR(tyP0936Trav.tyMotionStd.tyBtnJogRear.uiMaskRtStat));
		fUIInRtStatOff(ADR(tyP0936Trav.tyTrav.tyBtnGoToLaneA.uiMaskRtStat));
		fUIInRtStatOff(ADR(tyP0936Trav.tyTrav.tyBtnGoToLaneB.uiMaskRtStat));
		fUIInRtStatOff(ADR(tyP0936Trav.tyTrav.tyBtnGoToMag1.uiMaskRtStat));
		fUIInRtStatOff(ADR(tyP0936Trav.tyTrav.tyBtnGoToMag2.uiMaskRtStat));
		fUIInRtStatOff(ADR(tyP0936Trav.tyTrav.tyBtnGoToMag3.uiMaskRtStat));

	ELSIF tyP0936Trav.tyMotionStd.tyBtnJogRear.bRtCompl = TRUE OR tyP0936Trav.tyMotionStd.tyBtnJogRear.bValue = TRUE THEN
		fUIInRtStatOff(ADR(tyP0936Trav.tyMotionStd.tyBtnOrigin.uiMaskRtStat));
		fUIInRtStatOff(ADR(tyP0936Trav.tyMotionStd.tyBtnMovAbs.uiMaskRtStat));
		fUIInRtStatOff(ADR(tyP0936Trav.tyMotionStd.tyBtnMovRel.uiMaskRtStat));
		fUIInRtStatOff(ADR(tyP0936Trav.tyMotionStd.tyBtnJogFront.uiMaskRtStat));
		fUIInRtStatOff(ADR(tyP0936Trav.tyTrav.tyBtnGoToLaneA.uiMaskRtStat));
		fUIInRtStatOff(ADR(tyP0936Trav.tyTrav.tyBtnGoToLaneB.uiMaskRtStat));
		fUIInRtStatOff(ADR(tyP0936Trav.tyTrav.tyBtnGoToMag1.uiMaskRtStat));
		fUIInRtStatOff(ADR(tyP0936Trav.tyTrav.tyBtnGoToMag2.uiMaskRtStat));
		fUIInRtStatOff(ADR(tyP0936Trav.tyTrav.tyBtnGoToMag3.uiMaskRtStat));

	ELSIF tyP0936Trav.tyMotionStd.tyBtnJogFront.bRtCompl = TRUE OR tyP0936Trav.tyMotionStd.tyBtnJogFront.bValue = TRUE THEN
		fUIInRtStatOff(ADR(tyP0936Trav.tyMotionStd.tyBtnOrigin.uiMaskRtStat));
		fUIInRtStatOff(ADR(tyP0936Trav.tyMotionStd.tyBtnMovAbs.uiMaskRtStat));
		fUIInRtStatOff(ADR(tyP0936Trav.tyMotionStd.tyBtnMovRel.uiMaskRtStat));
		fUIInRtStatOff(ADR(tyP0936Trav.tyMotionStd.tyBtnJogRear.uiMaskRtStat));
		fUIInRtStatOff(ADR(tyP0936Trav.tyTrav.tyBtnGoToLaneA.uiMaskRtStat));
		fUIInRtStatOff(ADR(tyP0936Trav.tyTrav.tyBtnGoToLaneB.uiMaskRtStat));
		fUIInRtStatOff(ADR(tyP0936Trav.tyTrav.tyBtnGoToMag1.uiMaskRtStat));
		fUIInRtStatOff(ADR(tyP0936Trav.tyTrav.tyBtnGoToMag2.uiMaskRtStat));
		fUIInRtStatOff(ADR(tyP0936Trav.tyTrav.tyBtnGoToMag3.uiMaskRtStat));

	ELSIF tyP0936Trav.tyTrav.tyBtnGoToLaneA.bRtCompl = TRUE THEN
		fUIInRtStatOff(ADR(tyP0936Trav.tyMotionStd.tyBtnOrigin.uiMaskRtStat));
		fUIInRtStatOff(ADR(tyP0936Trav.tyMotionStd.tyBtnMovAbs.uiMaskRtStat));
		fUIInRtStatOff(ADR(tyP0936Trav.tyMotionStd.tyBtnMovRel.uiMaskRtStat));
		fUIInRtStatOff(ADR(tyP0936Trav.tyMotionStd.tyBtnJogFront.uiMaskRtStat));
		fUIInRtStatOff(ADR(tyP0936Trav.tyMotionStd.tyBtnJogRear.uiMaskRtStat));
		fUIInRtStatOff(ADR(tyP0936Trav.tyTrav.tyBtnGoToLaneB.uiMaskRtStat));
		fUIInRtStatOff(ADR(tyP0936Trav.tyTrav.tyBtnGoToMag1.uiMaskRtStat));
		fUIInRtStatOff(ADR(tyP0936Trav.tyTrav.tyBtnGoToMag2.uiMaskRtStat));
		fUIInRtStatOff(ADR(tyP0936Trav.tyTrav.tyBtnGoToMag3.uiMaskRtStat));

	ELSIF tyP0936Trav.tyTrav.tyBtnGoToLaneB.bRtCompl = TRUE THEN
		fUIInRtStatOff(ADR(tyP0936Trav.tyMotionStd.tyBtnOrigin.uiMaskRtStat));
		fUIInRtStatOff(ADR(tyP0936Trav.tyMotionStd.tyBtnMovAbs.uiMaskRtStat));
		fUIInRtStatOff(ADR(tyP0936Trav.tyMotionStd.tyBtnMovRel.uiMaskRtStat));
		fUIInRtStatOff(ADR(tyP0936Trav.tyMotionStd.tyBtnJogFront.uiMaskRtStat));
		fUIInRtStatOff(ADR(tyP0936Trav.tyMotionStd.tyBtnJogRear.uiMaskRtStat));
		fUIInRtStatOff(ADR(tyP0936Trav.tyTrav.tyBtnGoToLaneA.uiMaskRtStat));
		fUIInRtStatOff(ADR(tyP0936Trav.tyTrav.tyBtnGoToMag1.uiMaskRtStat));
		fUIInRtStatOff(ADR(tyP0936Trav.tyTrav.tyBtnGoToMag2.uiMaskRtStat));
		fUIInRtStatOff(ADR(tyP0936Trav.tyTrav.tyBtnGoToMag3.uiMaskRtStat));

	ELSIF tyP0936Trav.tyTrav.tyBtnGoToMag1.bRtCompl = TRUE THEN
		fUIInRtStatOff(ADR(tyP0936Trav.tyMotionStd.tyBtnOrigin.uiMaskRtStat));
		fUIInRtStatOff(ADR(tyP0936Trav.tyMotionStd.tyBtnMovAbs.uiMaskRtStat));
		fUIInRtStatOff(ADR(tyP0936Trav.tyMotionStd.tyBtnMovRel.uiMaskRtStat));
		fUIInRtStatOff(ADR(tyP0936Trav.tyMotionStd.tyBtnJogFront.uiMaskRtStat));
		fUIInRtStatOff(ADR(tyP0936Trav.tyMotionStd.tyBtnJogRear.uiMaskRtStat));
		fUIInRtStatOff(ADR(tyP0936Trav.tyTrav.tyBtnGoToLaneA.uiMaskRtStat));
		fUIInRtStatOff(ADR(tyP0936Trav.tyTrav.tyBtnGoToLaneB.uiMaskRtStat));
		fUIInRtStatOff(ADR(tyP0936Trav.tyTrav.tyBtnGoToMag2.uiMaskRtStat));
		fUIInRtStatOff(ADR(tyP0936Trav.tyTrav.tyBtnGoToMag3.uiMaskRtStat));

	ELSIF tyP0936Trav.tyTrav.tyBtnGoToMag2.bRtCompl = TRUE THEN
		fUIInRtStatOff(ADR(tyP0936Trav.tyMotionStd.tyBtnOrigin.uiMaskRtStat));
		fUIInRtStatOff(ADR(tyP0936Trav.tyMotionStd.tyBtnMovAbs.uiMaskRtStat));
		fUIInRtStatOff(ADR(tyP0936Trav.tyMotionStd.tyBtnMovRel.uiMaskRtStat));
		fUIInRtStatOff(ADR(tyP0936Trav.tyMotionStd.tyBtnJogFront.uiMaskRtStat));
		fUIInRtStatOff(ADR(tyP0936Trav.tyMotionStd.tyBtnJogRear.uiMaskRtStat));
		fUIInRtStatOff(ADR(tyP0936Trav.tyTrav.tyBtnGoToLaneA.uiMaskRtStat));
		fUIInRtStatOff(ADR(tyP0936Trav.tyTrav.tyBtnGoToLaneB.uiMaskRtStat));
		fUIInRtStatOff(ADR(tyP0936Trav.tyTrav.tyBtnGoToMag1.uiMaskRtStat));
		fUIInRtStatOff(ADR(tyP0936Trav.tyTrav.tyBtnGoToMag3.uiMaskRtStat));

	ELSIF tyP0936Trav.tyTrav.tyBtnGoToMag3.bRtCompl = TRUE THEN
		fUIInRtStatOff(ADR(tyP0936Trav.tyMotionStd.tyBtnOrigin.uiMaskRtStat));
		fUIInRtStatOff(ADR(tyP0936Trav.tyMotionStd.tyBtnMovAbs.uiMaskRtStat));
		fUIInRtStatOff(ADR(tyP0936Trav.tyMotionStd.tyBtnMovRel.uiMaskRtStat));
		fUIInRtStatOff(ADR(tyP0936Trav.tyMotionStd.tyBtnJogFront.uiMaskRtStat));
		fUIInRtStatOff(ADR(tyP0936Trav.tyMotionStd.tyBtnJogRear.uiMaskRtStat));
		fUIInRtStatOff(ADR(tyP0936Trav.tyTrav.tyBtnGoToLaneA.uiMaskRtStat));
		fUIInRtStatOff(ADR(tyP0936Trav.tyTrav.tyBtnGoToLaneB.uiMaskRtStat));
		fUIInRtStatOff(ADR(tyP0936Trav.tyTrav.tyBtnGoToMag1.uiMaskRtStat));
		fUIInRtStatOff(ADR(tyP0936Trav.tyTrav.tyBtnGoToMag2.uiMaskRtStat));

	END_IF

	//Axis Error
	IF tyP0936Trav.tyMotionStd.tyBtnPwr.bRtCompl = TRUE THEN
		fUIInRtStatOff(ADR(tyP0936Trav.tyMotionStd.tyBtnRst.uiMaskRtStat));
	ELSE
		fUIInRtStatHide(ADR(tyP0936Trav.tyMotionStd.tyBtnRst.uiMaskRtStat));
	END_IF

END_ACTION
```

#### Act_OptP0936UpdtDat.st
```iecst
ACTION Act_OptP0936UpdtDat:

	tyP0936Trav.tyMotionStd.tyNumCurrPos.diValue		:= p_diTravActualPos;
	tyP0936Trav.tyMotionStd.tyNumErrCode.diValue		:= UDINT_TO_DINT(p_udiTravAxisErrID);
	tyP0936Trav.tyMotionStd.tyBitmapPwr.usiValueIdx		:= BOOL_TO_USINT(p_bTravPwrOn);
	tyP0936Trav.tyMotionStd.tyBitmapRst.usiValueIdx		:= BOOL_TO_USINT(NOT p_bTravAxisErr);
	tyP0936Trav.tyMotionStd.tyBitmapOrigin.usiValueIdx	:= BOOL_TO_USINT(p_bTravIsHomed);
	tyP0936Trav.tyMotionStd.tyBtnFrontLmtSen.bValue		:= p_bTravFrontSen;
	tyP0936Trav.tyMotionStd.tyBtnRearLmtSen.bValue		:= p_bTravRearSen;

	//Machine Bitmap
	IF p_bTravIsHomed = TRUE THEN
		IF p_diTravActualPos <= (p_tyNtParamCurr.tyUITravTargetPos.diMax / 3) THEN
			tyP0936Trav.tyMotionStd.tyBitmapMc.uiValueIdx 	:= 5;
		ELSIF p_diTravActualPos <= (p_tyNtParamCurr.tyUITravTargetPos.diMax / 3 * 2) THEN
			tyP0936Trav.tyMotionStd.tyBitmapMc.uiValueIdx 	:= 6;
		ELSE
			tyP0936Trav.tyMotionStd.tyBitmapMc.uiValueIdx 	:= 7;
		END_IF
	ELSE
		tyP0936Trav.tyMotionStd.tyBitmapMc.uiValueIdx	:= 5;
	END_IF

	IF p_tyNtParamCurr.eProjMag = ULMagDual THEN
		IF p_tyNtParamCurr.bProjLifterMagPlatform AND p_tyNtParamCurr.bUIConvDirRL THEN
			IF 	tyP0936Trav.tyMotionStd.tyBitmapMc.uiValueIdx < 700 THEN
				tyP0936Trav.tyMotionStd.tyBitmapMc.uiValueIdx	:= tyP0936Trav.tyMotionStd.tyBitmapMc.uiValueIdx + 700;
			END_IF
		ELSIF p_tyNtParamCurr.bProjLifterMagPlatform THEN
			IF 	tyP0936Trav.tyMotionStd.tyBitmapMc.uiValueIdx < 600 THEN
				tyP0936Trav.tyMotionStd.tyBitmapMc.uiValueIdx	:= tyP0936Trav.tyMotionStd.tyBitmapMc.uiValueIdx + 600;
			END_IF
		ELSIF p_tyNtParamCurr.bMagAutoVerifyPrep = FALSE THEN
			IF 	tyP0936Trav.tyMotionStd.tyBitmapMc.uiValueIdx < 100 THEN
				tyP0936Trav.tyMotionStd.tyBitmapMc.uiValueIdx	:= tyP0936Trav.tyMotionStd.tyBitmapMc.uiValueIdx + 300;
			END_IF
		ELSE
			IF 	tyP0936Trav.tyMotionStd.tyBitmapMc.uiValueIdx < 300 THEN
				tyP0936Trav.tyMotionStd.tyBitmapMc.uiValueIdx	:= tyP0936Trav.tyMotionStd.tyBitmapMc.uiValueIdx + 300;
			END_IF
		END_IF
	ELSIF p_tyNtParamCurr.eProjMag = ULMagTriple THEN
		IF p_tyNtParamCurr.bProjLifterMagPlatform AND p_tyNtParamCurr.bUIConvDirRL THEN
			IF 	tyP0936Trav.tyMotionStd.tyBitmapMc.uiValueIdx < 800 THEN
				tyP0936Trav.tyMotionStd.tyBitmapMc.uiValueIdx	:= tyP0936Trav.tyMotionStd.tyBitmapMc.uiValueIdx + 800;
			END_IF
		ELSIF p_tyNtParamCurr.bProjLifterMagPlatform THEN
			IF 	tyP0936Trav.tyMotionStd.tyBitmapMc.uiValueIdx < 500 THEN
				tyP0936Trav.tyMotionStd.tyBitmapMc.uiValueIdx	:= tyP0936Trav.tyMotionStd.tyBitmapMc.uiValueIdx + 500;
			END_IF
		ELSIF  p_tyNtParamCurr.bProjMotorizedPusherPrep = FALSE THEN//p_tyNtParamCurr.bMagAutoVerifyPrep = TRUE AND p_tyNtParamCurr.bProjMotorizedPusherPrep = FALSE THEN
			IF 	tyP0936Trav.tyMotionStd.tyBitmapMc.uiValueIdx < 200 THEN
				tyP0936Trav.tyMotionStd.tyBitmapMc.uiValueIdx	:= tyP0936Trav.tyMotionStd.tyBitmapMc.uiValueIdx + 200;
			END_IF
		ELSIF  p_tyNtParamCurr.bMagAutoVerifyPrep = FALSE AND p_tyNtParamCurr.bProjMotorizedPusherPrep = TRUE THEN
			IF 	tyP0936Trav.tyMotionStd.tyBitmapMc.uiValueIdx < 400 AND p_tyNtParamCurr.bCurtainSenPrep THEN
				tyP0936Trav.tyMotionStd.tyBitmapMc.uiValueIdx	:= tyP0936Trav.tyMotionStd.tyBitmapMc.uiValueIdx + 440;
			ELSE
				tyP0936Trav.tyMotionStd.tyBitmapMc.uiValueIdx	:= tyP0936Trav.tyMotionStd.tyBitmapMc.uiValueIdx + 400;
			END_IF
		END_IF
	END_IF

END_ACTION
```

#### Act_OptP0936Keypad.st
```iecst
ACTION Act_OptP0936Keypad:

	IF fUIOutRtStatTPIsOpen(ADR(tyP0936Trav.tyMotionStd.tyNumTargetPos.uiRtStat)) = TRUE THEN
		tyProperty.tyKeypad.tyStringTitle.sKeypadTitle		:= tyP0936Trav.tyMotionStd.tyNumTargetPos.sKeypadTitle;

	ELSIF fUIOutRtStatTPIsOpen(ADR(tyP0936Trav.tyMotionStd.tyNumStepSize.uiRtStat)) = TRUE THEN
		tyProperty.tyKeypad.tyStringTitle.sKeypadTitle		:= tyP0936Trav.tyMotionStd.tyNumStepSize.sKeypadTitle;

	ELSIF fUIOutRtStatTPIsOpen(ADR(tyP0936Trav.tyMotionStd.tyNumNomSpd.uiRtStat)) = TRUE THEN
		tyProperty.tyKeypad.tyStringTitle.sKeypadTitle		:= tyP0936Trav.tyMotionStd.tyNumNomSpd.sKeypadTitle;

	ELSIF fUIOutRtStatTPIsOpen(ADR(tyP0936Trav.tyMotionStd.tyNumSlwSpd.uiRtStat)) = TRUE THEN
		tyProperty.tyKeypad.tyStringTitle.sKeypadTitle		:= tyP0936Trav.tyMotionStd.tyNumSlwSpd.sKeypadTitle;

	END_IF

END_ACTION
```

#### Act_OptP0936RstMnl.st
```iecst
ACTION Act_OptP0936RstMnl:

	IF EDGEPOS((bManualMod = FALSE) OR (p_eTravStatus = Error)) THEN

		eTravAct	:= TravActIdle;

		bJogSlow				:= FALSE;
		bJogFast				:= FALSE;
		fbJogSlowToFastDlyTm.IN	:= FALSE;

		tyP0936Trav.tyTrav.tyBtnGoToLaneA.bRtCompl				:= FALSE;
		tyP0936Trav.tyTrav.tyBtnGoToLaneA.bValue				:= FALSE;
		tyP0936Trav.tyTrav.tyBtnGoToLaneA.bRtLk					:= FALSE;
		tyP0936Trav.tyTrav.tyBtnGoToLaneA.uiMaskRtStat.0		:= FALSE;

		tyP0936Trav.tyTrav.tyBtnGoToLaneB.bRtCompl				:= FALSE;
		tyP0936Trav.tyTrav.tyBtnGoToLaneB.bValue				:= FALSE;
		tyP0936Trav.tyTrav.tyBtnGoToLaneB.bRtLk					:= FALSE;
		tyP0936Trav.tyTrav.tyBtnGoToLaneB.uiMaskRtStat.0		:= FALSE;

		tyP0936Trav.tyTrav.tyBtnGoToMag1.bRtCompl				:= FALSE;
		tyP0936Trav.tyTrav.tyBtnGoToMag1.bValue					:= FALSE;
		tyP0936Trav.tyTrav.tyBtnGoToMag1.bRtLk					:= FALSE;
		tyP0936Trav.tyTrav.tyBtnGoToMag1.uiMaskRtStat.0			:= FALSE;

		tyP0936Trav.tyTrav.tyBtnGoToMag2.bRtCompl				:= FALSE;
		tyP0936Trav.tyTrav.tyBtnGoToMag2.bValue					:= FALSE;
		tyP0936Trav.tyTrav.tyBtnGoToMag2.bRtLk					:= FALSE;
		tyP0936Trav.tyTrav.tyBtnGoToMag2.uiMaskRtStat.0			:= FALSE;

		tyP0936Trav.tyTrav.tyBtnGoToMag3.bRtCompl				:= FALSE;
		tyP0936Trav.tyTrav.tyBtnGoToMag3.bValue					:= FALSE;
		tyP0936Trav.tyTrav.tyBtnGoToMag3.bRtLk					:= FALSE;
		tyP0936Trav.tyTrav.tyBtnGoToMag3.uiMaskRtStat.0			:= FALSE;

		tyP0936Trav.tyMotionStd.tyBtnPwr.bRtCompl				:= FALSE;
		tyP0936Trav.tyMotionStd.tyBtnStop.bRtCompl				:= FALSE;
		tyP0936Trav.tyMotionStd.tyBtnOrigin.bRtCompl			:= FALSE;
		tyP0936Trav.tyMotionStd.tyBtnRst.bRtCompl				:= FALSE;
		tyP0936Trav.tyMotionStd.tyBtnMovAbs.bRtCompl			:= FALSE;
		tyP0936Trav.tyMotionStd.tyBtnMovRel.bRtCompl			:= FALSE;
		tyP0936Trav.tyMotionStd.tyBtnJogFront.bRtCompl			:= FALSE;
		tyP0936Trav.tyMotionStd.tyBtnJogRear.bRtCompl			:= FALSE;

		tyP0936Trav.tyMotionStd.tyBtnPwr.bValue					:= FALSE;
		tyP0936Trav.tyMotionStd.tyBtnStop.bValue				:= TRUE;
		tyP0936Trav.tyMotionStd.tyBtnOrigin.bValue				:= FALSE;
		tyP0936Trav.tyMotionStd.tyBtnRst.bValue					:= FALSE;
		tyP0936Trav.tyMotionStd.tyBtnMovAbs.bValue				:= FALSE;
		tyP0936Trav.tyMotionStd.tyBtnMovRel.bValue				:= FALSE;
		tyP0936Trav.tyMotionStd.tyBtnJogFront.bValue			:= FALSE;
		tyP0936Trav.tyMotionStd.tyBtnJogRear.bValue				:= FALSE;

		tyP0936Trav.tyMotionStd.tyBtnPwr.bRtLk					:= FALSE;
		tyP0936Trav.tyMotionStd.tyBtnStop.bRtLk					:= TRUE;
		tyP0936Trav.tyMotionStd.tyBtnOrigin.bRtLk				:= FALSE;
		tyP0936Trav.tyMotionStd.tyBtnRst.bRtLk					:= FALSE;
		tyP0936Trav.tyMotionStd.tyBtnMovAbs.bRtLk				:= FALSE;
		tyP0936Trav.tyMotionStd.tyBtnMovRel.bRtLk				:= FALSE;
		tyP0936Trav.tyMotionStd.tyBtnJogFront.bRtLk				:= FALSE;
		tyP0936Trav.tyMotionStd.tyBtnJogRear.bRtLk				:= FALSE;

		tyP0936Trav.tyMotionStd.tyBtnPwr.uiMaskRtStat			:= TRUE;
		tyP0936Trav.tyMotionStd.tyBtnOrigin.uiMaskRtStat		:= FALSE;
		tyP0936Trav.tyMotionStd.tyBtnRst.uiMaskRtStat			:= TRUE;
		tyP0936Trav.tyMotionStd.tyBtnMovAbs.uiMaskRtStat		:= FALSE;
		tyP0936Trav.tyMotionStd.tyBtnMovRel.uiMaskRtStat		:= FALSE;
		tyP0936Trav.tyMotionStd.tyBtnJogFront.uiMaskRtStat		:= FALSE;
		tyP0936Trav.tyMotionStd.tyBtnJogRear.uiMaskRtStat		:= FALSE;

	END_IF

	eInShutterAct	:= PneuActIdle;
	eOutShutterAct	:= PneuActIdle;

	tyP0936Trav.tyInOutletShutterFB.tyBtnClose.bRtCompl	:= FALSE;
	tyP0936Trav.tyInOutletShutterFB.tyBtnClose.bValue	:= FALSE;
	tyP0936Trav.tyInOutletShutterFB.tyBtnOpen.bRtCompl	:= FALSE;
	tyP0936Trav.tyInOutletShutterFB.tyBtnOpen.bValue	:= FALSE;

END_ACTION
```

#### Act_EntP0937Disp.st
```iecst
ACTION Act_EntP0937Disp:

	// Access Address
	p_tyC0001MotionStd ACCESS ADR(tyP0937AWPushOrPuller.tyMotionStd);

	p_tyC0002FullMask ACCESS ADR(tyP0937AWPushOrPuller.tyFullMaskHide);

	p_tyC0004Navi ACCESS ADR(tyP0937AWPushOrPuller.tyNaviBack);

	p_tyC0005Main ACCESS ADR(tyCommon.tyMain);

	p_tyC0007Notif ACCESS ADR(tyCommon.tyNotif);

	p_tyC0008MsgBox ACCESS ADR(tyP0937AWPushOrPuller.tyMsgBoxHide);

	p_tyC0009Info ACCESS ADR(tyCommon.tyInfo);

	p_tyP0937AWPushOrPuller ACCESS ADR(tyP0937AWPushOrPuller.tyAW);

	p_tyP0937InOutletShutterFB ACCESS ADR(tyP0937AWPushOrPuller.tyInOutletShutterFB);

	// Display
	tyP0937AWPushOrPuller.tyAW.tyNumNewWidth.diValue		:= p_tyProdRcpCurrRcp0.diWidthInUM;

	tyP0937AWPushOrPuller.tyMotionStd.tyBtnPwr.bValue		:= p_bAWPushOrPullerPwrOn;

	fbLmtRstTm(IN := FALSE);

END_ACTION
```

#### Act_OptP0937Navi.st
```iecst
ACTION Act_OptP0937Navi:

IF tyP0937AWPushOrPuller.tyNaviBack.tyBtnBack.bRtCompl = TRUE THEN
	tyP0937AWPushOrPuller.tyNaviBack.tyBtnBack.bRtCompl		:= FALSE;
	tyP0937AWPushOrPuller.tyNaviBack.tyBtnBack.bValue		:= FALSE;

	eChgPage		:= UIP0920MtrNPneuCtrl;
END_IF

END_ACTION
```

#### Act_OptP0937FullMask.st
```iecst
ACTION Act_OptP0937FullMask:

	IF eCurrPage = UIP0937AWPushOrPuller THEN

		IF p_tyDI.bEStopSig = FALSE THEN
			p_tyC0002FullMask ACCESS ADR(tyP0934AW.tyFullMaskEStop);

		ELSIF p_tyDI.bCoverSWSig = FALSE THEN
			p_tyC0002FullMask ACCESS ADR(tyP0934AW.tyFullMaskCWSig);

		ELSIF p_tyDI.bSafetyRlySig = FALSE THEN
			p_tyC0002FullMask ACCESS ADR(tyP0934AW.tyFullMaskSafetyRly);

		ELSIF p_tyDI.bConvLftSen THEN
			p_tyC0002FullMask ACCESS ADR(tyP0934AW.tyFullMaskLftSenInterrupt);

		ELSIF p_tyDI.bConvRgtSen THEN
			p_tyC0002FullMask ACCESS ADR(tyP0934AW.tyFullMaskRgtSenInterrupt);

		ELSIF (p_tyNtParamCurr.bProjInletShutPrep AND p_tyDI.bInShutterCloseRS = FALSE) AND NOT(bBypassShutForCalib) THEN
			p_tyC0002FullMask ACCESS ADR(tyP0934AW.tyFullMaskInShutOpnInterrupt);

		ELSIF ((p_tyDI.bOutShutterCloseRS = FALSE AND p_tyNtParamCurr.bProjOutletShutPrep) OR (p_tyDI.bOutShutterCloseRS2 = FALSE AND p_tyNtParamCurr.bProjOutletShut2Prep )OR (p_tyDI.bOutShutterCloseRS3 = FALSE AND p_tyNtParamCurr.bProjOutletShut3Prep)) AND NOT(bBypassShutForCalib) THEN
			IF p_tyNtParamCurr.bCurtainSenPrep THEN
				IF (p_tyDI.bOutShutterCloseRS = FALSE AND p_tyNtParamCurr.bProjOutletShutPrep) OR (p_tyDI.bOutShutterCloseRS2 = FALSE AND p_tyNtParamCurr.bProjOutletShut2Prep)OR (p_tyDI.bOutShutterCloseRS3 = FALSE AND p_tyNtParamCurr.bProjOutletShut3Prep )THEN
					p_tyC0002FullMask ACCESS ADR(tyP0934AW.tyFullMaskOutShutOpnInterrupt);
				END_IF
			ELSE
				IF p_tyDI.bOutShutterCloseRS = FALSE THEN
					p_tyC0002FullMask ACCESS ADR(tyP0934AW.tyFullMaskOutShutOpnInterrupt);
				END_IF
			END_IF
		ELSE
			p_tyC0002FullMask ACCESS ADR(tyP0934AW.tyFullMaskHide);

		END_IF

	END_IF

END_ACTION
```

#### Act_OptP0937FBCtrl.st
```iecst
ACTION Act_OptP0937FBCtrl:

	fbJogSlowToFastDlyTm.PT			:= T#2s;
	fbJogSlowToFastDlyTm;
	fbLmtRstTm;

	//Conveyor Sensor Interruption
	IF p_tyDI.bPusherRetRS = FALSE THEN
		tyP0937AWPushOrPuller.tyMotionStd.tyBtnStop.bRtCompl	:= TRUE;
	END_IF

//	IF EDGEPOS((p_udiAWPushOrPullerAxisErrID = 21570 OR p_udiAWPushOrPullerAxisErrID = 21571)
	IF EDGEPOS ((p_bAWPushOrPullerFwdLmtSen OR p_bAWPushOrPullerRevLmtSen)
		AND tyP0937AWPushOrPuller.tyMotionStd.tyBtnJogOpen.bValue = FALSE
		AND tyP0937AWPushOrPuller.tyMotionStd.tyBtnJogClose.bValue = FALSE)
	THEN
		fbLmtRstTm.IN	:= TRUE;
	END_IF

	IF fbLmtRstTm.Q = TRUE THEN
		tyP0937AWPushOrPuller.tyMotionStd.tyBtnRst.bRtCompl		:= TRUE;
	END_IF

	IF (tyP0937AWPushOrPuller.tyMotionStd.tyBtnJogOpen.bValue = FALSE AND tyP0937AWPushOrPuller.tyMotionStd.tyBtnJogClose.bValue = FALSE) AND (p_bAWPushOrPullerJogging = TRUE) THEN
		bJogStopAWPushOrPuller	:= TRUE;
	END_IF

	IF tyP0937AWPushOrPuller.tyMotionStd.tyBtnStop.bRtCompl = TRUE THEN
		eAWPushOrPullerAct		:= AWActStop;

		IF p_eAWPushOrPullerStat = AWActStop AND p_eAWPushOrPullerStatus = Done THEN
			eAWPushOrPullerAct	:= AWActIdle;

			tyP0937AWPushOrPuller.tyMotionStd.tyBtnStop.bRtCompl	:= FALSE;
			tyP0937AWPushOrPuller.tyMotionStd.tyBtnJogOpen.bRtCompl	:= FALSE;
			tyP0937AWPushOrPuller.tyMotionStd.tyBtnJogClose.bRtCompl:= FALSE;
			tyP0937AWPushOrPuller.tyMotionStd.tyBtnOrigin.bRtCompl	:= FALSE;
			tyP0937AWPushOrPuller.tyMotionStd.tyBtnMovAbs.bRtCompl	:= FALSE;
			tyP0937AWPushOrPuller.tyMotionStd.tyBtnMovRel.bRtCompl	:= FALSE;
			tyP0937AWPushOrPuller.tyAW.tyBtnGo.bRtCompl				:= FALSE;

			tyP0937AWPushOrPuller.tyMotionStd.tyBtnStop.bValue		:= TRUE;
			tyP0937AWPushOrPuller.tyMotionStd.tyBtnJogOpen.bValue	:= FALSE;
			tyP0937AWPushOrPuller.tyMotionStd.tyBtnJogClose.bValue	:= FALSE;
			tyP0937AWPushOrPuller.tyMotionStd.tyBtnOrigin.bValue	:= FALSE;
			tyP0937AWPushOrPuller.tyMotionStd.tyBtnMovAbs.bValue	:= FALSE;
			tyP0937AWPushOrPuller.tyMotionStd.tyBtnMovRel.bValue	:= FALSE;
			tyP0937AWPushOrPuller.tyAW.tyBtnGo.bValue				:= FALSE;

			tyP0937AWPushOrPuller.tyMotionStd.tyBtnStop.bRtLk		:= TRUE;
			tyP0937AWPushOrPuller.tyMotionStd.tyBtnJogOpen.bRtLk	:= FALSE;
			tyP0937AWPushOrPuller.tyMotionStd.tyBtnJogClose.bRtLk	:= FALSE;
			tyP0937AWPushOrPuller.tyMotionStd.tyBtnOrigin.bRtLk		:= FALSE;
			tyP0937AWPushOrPuller.tyMotionStd.tyBtnMovAbs.bRtLk		:= FALSE;
			tyP0937AWPushOrPuller.tyMotionStd.tyBtnMovRel.bRtLk		:= FALSE;
			tyP0937AWPushOrPuller.tyAW.tyBtnGo.bRtLk				:= FALSE;
		END_IF

	ELSIF (tyP0937AWPushOrPuller.tyMotionStd.tyBtnJogOpen.bRtCompl = TRUE) OR (tyP0937AWPushOrPuller.tyMotionStd.tyBtnJogClose.bRtCompl = TRUE) OR (bJogStopAWPushOrPuller = TRUE) THEN
		bJogSlow					:= FALSE;
		bJogFast					:= FALSE;
		fbJogSlowToFastDlyTm.IN		:= FALSE;

		eAWPushOrPullerAct		:= AWActJogStop;

		IF p_eAWPushOrPullerStat = AWActJogStop AND p_eAWPushOrPullerStatus = Done THEN
			eAWPushOrPullerAct	:= AWActIdle;

			bJogStopAWPushOrPuller	:= FALSE;

			tyP0937AWPushOrPuller.tyMotionStd.tyBtnStop.bRtCompl	:= FALSE;
			tyP0937AWPushOrPuller.tyMotionStd.tyBtnJogOpen.bRtCompl	:= FALSE;
			tyP0937AWPushOrPuller.tyMotionStd.tyBtnJogClose.bRtCompl:= FALSE;
			tyP0937AWPushOrPuller.tyMotionStd.tyBtnOrigin.bRtCompl	:= FALSE;
			tyP0937AWPushOrPuller.tyMotionStd.tyBtnMovAbs.bRtCompl	:= FALSE;
			tyP0937AWPushOrPuller.tyMotionStd.tyBtnMovRel.bRtCompl	:= FALSE;
			tyP0937AWPushOrPuller.tyAW.tyBtnGo.bRtCompl				:= FALSE;

			tyP0937AWPushOrPuller.tyMotionStd.tyBtnStop.bValue		:= TRUE;
			tyP0937AWPushOrPuller.tyMotionStd.tyBtnJogOpen.bValue	:= FALSE;
			tyP0937AWPushOrPuller.tyMotionStd.tyBtnJogClose.bValue	:= FALSE;
			tyP0937AWPushOrPuller.tyMotionStd.tyBtnOrigin.bValue	:= FALSE;
			tyP0937AWPushOrPuller.tyMotionStd.tyBtnMovAbs.bValue	:= FALSE;
			tyP0937AWPushOrPuller.tyMotionStd.tyBtnMovRel.bValue	:= FALSE;
			tyP0937AWPushOrPuller.tyAW.tyBtnGo.bValue				:= FALSE;

			tyP0937AWPushOrPuller.tyMotionStd.tyBtnStop.bRtLk		:= TRUE;
			tyP0937AWPushOrPuller.tyMotionStd.tyBtnJogOpen.bRtLk	:= FALSE;
			tyP0937AWPushOrPuller.tyMotionStd.tyBtnJogClose.bRtLk	:= FALSE;
			tyP0937AWPushOrPuller.tyMotionStd.tyBtnOrigin.bRtLk		:= FALSE;
			tyP0937AWPushOrPuller.tyMotionStd.tyBtnMovAbs.bRtLk		:= FALSE;
			tyP0937AWPushOrPuller.tyMotionStd.tyBtnMovRel.bRtLk		:= FALSE;
			tyP0937AWPushOrPuller.tyAW.tyBtnGo.bRtLk				:= FALSE;
		END_IF

	ELSIF tyP0937AWPushOrPuller.tyMotionStd.tyBtnPwr.bRtCompl = TRUE THEN
		tyP0937AWPushOrPuller.tyMotionStd.tyBtnPwr.bRtLk	:= TRUE;

		IF tyP0937AWPushOrPuller.tyMotionStd.tyBtnPwr.bValue = TRUE THEN
			eAWPushOrPullerAct		:= AWActPwrOn;

			IF p_eAWPushOrPullerStat = AWActPwrOn AND p_eAWPushOrPullerStatus = Done THEN
				eAWPushOrPullerAct	:= AWActIdle;

				tyP0937AWPushOrPuller.tyMotionStd.tyBtnPwr.bRtCompl	:= FALSE;
				tyP0937AWPushOrPuller.tyMotionStd.tyBtnPwr.bRtLk		:= FALSE;
			END_IF
		ELSE
			eAWPushOrPullerAct	:= AWActPwrOff;

			IF p_eAWPushOrPullerStat = AWActPwrOff AND p_eAWPushOrPullerStatus = Done THEN
				eAWPushOrPullerAct	:= AWActIdle;

				tyP0937AWPushOrPuller.tyMotionStd.tyBtnPwr.bRtCompl			:= FALSE;
				tyP0937AWPushOrPuller.tyMotionStd.tyBtnPwr.bRtLk			:= FALSE;
			END_IF
		END_IF

	ELSIF tyP0937AWPushOrPuller.tyMotionStd.tyBtnOrigin.bRtCompl = TRUE THEN
		tyP0937AWPushOrPuller.tyMotionStd.tyBtnOrigin.bValue	:= TRUE;
		tyP0937AWPushOrPuller.tyMotionStd.tyBtnStop.bValue	:= FALSE;

		tyP0937AWPushOrPuller.tyMotionStd.tyBtnOrigin.bRtLk	:= TRUE;
		tyP0937AWPushOrPuller.tyMotionStd.tyBtnStop.bRtLk		:= FALSE;

		eAWPushOrPullerAct		:= AWActHoming;

		IF p_eAWPushOrPullerStat = AWActHoming AND p_eAWPushOrPullerStatus = Done THEN
			eAWPushOrPullerAct	:= AWActIdle;

			tyP0937AWPushOrPuller.tyMotionStd.tyBtnOrigin.bRtCompl	:= FALSE;
			tyP0937AWPushOrPuller.tyMotionStd.tyBtnOrigin.bValue		:= FALSE;
			tyP0937AWPushOrPuller.tyMotionStd.tyBtnStop.bValue		:= TRUE;

			tyP0937AWPushOrPuller.tyMotionStd.tyBtnOrigin.bRtLk		:= FALSE;
			tyP0937AWPushOrPuller.tyMotionStd.tyBtnStop.bRtLk			:= TRUE;
		END_IF

	ELSIF tyP0937AWPushOrPuller.tyMotionStd.tyBtnRst.bRtCompl = TRUE THEN
		tyP0937AWPushOrPuller.tyMotionStd.tyBtnRst.bValue					:= TRUE;
		tyP0937AWPushOrPuller.tyMotionStd.tyBtnRst.bRtLk					:= TRUE;

		eAWPushOrPullerAct		:= AWActRstAxisErr;

		IF p_eAWPushOrPullerStat = AWActRstAxisErr AND p_eAWPushOrPullerStatus = Done THEN
			eAWPushOrPullerAct	:= AWActIdle;

			tyP0937AWPushOrPuller.tyMotionStd.tyBtnRst.bRtCompl		:= FALSE;
			tyP0937AWPushOrPuller.tyMotionStd.tyBtnRst.bValue			:= FALSE;
			tyP0937AWPushOrPuller.tyMotionStd.tyBtnRst.bRtLk			:= FALSE;

			fbLmtRstTm.IN			:= FALSE;
		END_IF

	ELSIF tyP0937AWPushOrPuller.tyAW.tyBtnGo.bRtCompl = TRUE THEN
		tyP0937AWPushOrPuller.tyAW.tyBtnGo.bValue				:= TRUE;
		tyP0937AWPushOrPuller.tyMotionStd.tyBtnStop.bValue	:= FALSE;

		tyP0937AWPushOrPuller.tyAW.tyBtnGo.bRtLk				:= TRUE;
		tyP0937AWPushOrPuller.tyMotionStd.tyBtnStop.bRtLk		:= FALSE;

		diMnlAWPushOrPullerGoWidth	:= (tyP0937AWPushOrPuller.tyAW.tyNumNewWidth.diValue)/2;
		diMnlAWPushOrPullerNomSpd		:= tyP0937AWPushOrPuller.tyMotionStd.tyNumNomSpd.diValue;

		eAWPushOrPullerAct		:= AWActGoWidth;

		IF p_eAWPushOrPullerStat = AWActGoWidth AND p_eAWPushOrPullerStatus = Done THEN
			eAWPushOrPullerAct	:= AWActIdle;

			tyP0937AWPushOrPuller.tyAW.tyBtnGo.bRtCompl			:= FALSE;
			tyP0937AWPushOrPuller.tyAW.tyBtnGo.bValue				:= FALSE;
			tyP0937AWPushOrPuller.tyMotionStd.tyBtnStop.bValue	:= TRUE;

			tyP0937AWPushOrPuller.tyAW.tyBtnGo.bRtLk				:= FALSE;
			tyP0937AWPushOrPuller.tyMotionStd.tyBtnStop.bRtLk		:= TRUE;
		END_IF

	ELSIF tyP0937AWPushOrPuller.tyMotionStd.tyBtnMovAbs.bRtCompl = TRUE THEN
		tyP0937AWPushOrPuller.tyMotionStd.tyBtnMovAbs.bValue		:= TRUE;
		tyP0937AWPushOrPuller.tyMotionStd.tyBtnStop.bValue		:= FALSE;

		tyP0937AWPushOrPuller.tyMotionStd.tyBtnMovAbs.bRtLk		:= TRUE;
		tyP0937AWPushOrPuller.tyMotionStd.tyBtnStop.bRtLk			:= FALSE;

		diMnlAWPushOrPullerTargetPos	:= tyP0937AWPushOrPuller.tyMotionStd.tyNumTargetPos.diValue;
		diMnlAWPushOrPullerNomSpd		:= tyP0937AWPushOrPuller.tyMotionStd.tyNumNomSpd.diValue;

		eAWPushOrPullerAct		:= AWActMovAbs;

		IF p_eAWPushOrPullerStat = AWActMovAbs AND p_eAWPushOrPullerStatus = Done THEN
			eAWPushOrPullerAct	:= AWActIdle;

			tyP0937AWPushOrPuller.tyMotionStd.tyBtnMovAbs.bRtCompl	:= FALSE;
			tyP0937AWPushOrPuller.tyMotionStd.tyBtnMovAbs.bValue		:= FALSE;
			tyP0937AWPushOrPuller.tyMotionStd.tyBtnStop.bValue		:= TRUE;

			tyP0937AWPushOrPuller.tyMotionStd.tyBtnMovAbs.bRtLk		:= FALSE;
			tyP0937AWPushOrPuller.tyMotionStd.tyBtnStop.bRtLk			:= TRUE;
		END_IF

	ELSIF tyP0937AWPushOrPuller.tyMotionStd.tyBtnMovRel.bRtCompl = TRUE THEN
		tyP0937AWPushOrPuller.tyMotionStd.tyBtnMovRel.bValue			:= TRUE;
		tyP0937AWPushOrPuller.tyMotionStd.tyBtnStop.bValue			:= FALSE;

		tyP0937AWPushOrPuller.tyMotionStd.tyBtnMovRel.bRtLk			:= TRUE;
		tyP0937AWPushOrPuller.tyMotionStd.tyBtnStop.bRtLk				:= FALSE;

		diMnlAWPushOrPullerStepSize	:= tyP0937AWPushOrPuller.tyMotionStd.tyNumStepSize.diValue;
		diMnlAWPushOrPullerNomSpd		:= tyP0937AWPushOrPuller.tyMotionStd.tyNumNomSpd.diValue;

		eAWPushOrPullerAct		:= AWActMovRel;

		IF p_eAWPushOrPullerStat = AWActMovRel AND p_eAWPushOrPullerStatus = Done THEN
			eAWPushOrPullerAct	:= AWActIdle;

			tyP0937AWPushOrPuller.tyMotionStd.tyBtnMovRel.bRtCompl	:= FALSE;
			tyP0937AWPushOrPuller.tyMotionStd.tyBtnMovRel.bValue		:= FALSE;
			tyP0937AWPushOrPuller.tyMotionStd.tyBtnStop.bValue		:= TRUE;

			tyP0937AWPushOrPuller.tyMotionStd.tyBtnMovRel.bRtLk		:= FALSE;
			tyP0937AWPushOrPuller.tyMotionStd.tyBtnStop.bRtLk			:= TRUE;
		END_IF

	ELSIF (tyP0937AWPushOrPuller.tyMotionStd.tyBtnJogOpen.bValue = TRUE) AND (fbJogSlowToFastDlyTm.Q = FALSE) AND (bJogSlow = FALSE) THEN
		tyP0937AWPushOrPuller.tyMotionStd.tyBtnStop.bValue		:= FALSE;
		tyP0937AWPushOrPuller.tyMotionStd.tyBtnStop.bRtLk			:= FALSE;

		fbJogSlowToFastDlyTm.IN	:= TRUE;

		diMnlAWPushOrPullerJogSpd		:= tyP0937AWPushOrPuller.tyMotionStd.tyNumSlwSpd.diValue;

		eAWPushOrPullerAct		:= AWActJogOpen;

		IF p_eAWPushOrPullerStat = AWActJogOpen AND p_eAWPushOrPullerStatus = Done THEN
			eAWPushOrPullerAct	:= AWActIdle;
			bJogSlow		:= TRUE;
		ELSIF p_eAWPushOrPullerStatus = Error THEN
			fbJogSlowToFastDlyTm.IN	:= FALSE;
			bJogSlow		:= TRUE;
		END_IF

	ELSIF (tyP0937AWPushOrPuller.tyMotionStd.tyBtnJogOpen.bValue = TRUE) AND (fbJogSlowToFastDlyTm.Q = TRUE) AND (bJogFast = FALSE) THEN
		tyP0937AWPushOrPuller.tyMotionStd.tyBtnStop.bValue	:= FALSE;
		tyP0937AWPushOrPuller.tyMotionStd.tyBtnStop.bRtLk		:= FALSE;

		fbJogSlowToFastDlyTm.IN		:= TRUE;

		diMnlAWPushOrPullerJogSpd		:= tyP0937AWPushOrPuller.tyMotionStd.tyNumNomSpd.diValue;

		eAWPushOrPullerAct	:= AWActJogOpen;

		IF p_eAWPushOrPullerStat = AWActJogOpen AND p_eAWPushOrPullerStatus = Done THEN
			eAWPushOrPullerAct	:= AWActIdle;
			bJogFast				:= TRUE;
		ELSIF p_eAWPushOrPullerStatus = Error THEN
			fbJogSlowToFastDlyTm.IN	:= FALSE;
			bJogFast				:= TRUE;
		END_IF

	ELSIF (tyP0937AWPushOrPuller.tyMotionStd.tyBtnJogClose.bValue = TRUE) AND (fbJogSlowToFastDlyTm.Q = FALSE) AND (bJogSlow = FALSE) THEN
		tyP0937AWPushOrPuller.tyMotionStd.tyBtnStop.bValue					:= FALSE;
		tyP0937AWPushOrPuller.tyMotionStd.tyBtnStop.bRtLk					:= FALSE;

		fbJogSlowToFastDlyTm.IN		:= TRUE;

		diMnlAWPushOrPullerJogSpd		:= tyP0937AWPushOrPuller.tyMotionStd.tyNumSlwSpd.diValue;

		eAWPushOrPullerAct		:= AWActJogClose;

		IF p_eAWPushOrPullerStat = AWActJogClose AND p_eAWPushOrPullerStatus = Done THEN
			eAWPushOrPullerAct	:= AWActIdle;
			bJogSlow				:= TRUE;
		ELSIF p_eAWPushOrPullerStatus = Error THEN
			fbJogSlowToFastDlyTm.IN	:= FALSE;
			bJogSlow				:= TRUE;
		END_IF

	ELSIF (tyP0937AWPushOrPuller.tyMotionStd.tyBtnJogClose.bValue = TRUE) AND (fbJogSlowToFastDlyTm.Q = TRUE) AND (bJogFast = FALSE) THEN
		tyP0937AWPushOrPuller.tyMotionStd.tyBtnStop.bValue	:= FALSE;
		tyP0937AWPushOrPuller.tyMotionStd.tyBtnStop.bRtLk		:= FALSE;

		fbJogSlowToFastDlyTm.IN		:= TRUE;

		diMnlAWPushOrPullerJogSpd		:= tyP0937AWPushOrPuller.tyMotionStd.tyNumNomSpd.diValue;

		eAWPushOrPullerAct			:= AWActJogClose;

		IF p_eAWPushOrPullerStat = AWActJogClose AND p_eAWPushOrPullerStatus = Done THEN
			eAWPushOrPullerAct	:= AWActIdle;
			bJogFast				:= TRUE;
		ELSIF p_eAWPushOrPullerStatus = Error THEN
			fbJogSlowToFastDlyTm.IN	:= FALSE;
			bJogFast				:= TRUE;
		END_IF

	END_IF

END_ACTION
```

#### Act_OptP0937FBStat.st
```iecst
ACTION Act_OptP0937FBStat:

	IF p_bAWPushOrPullerAxisErr = TRUE THEN
		tyP0937AWPushOrPuller.tyMotionStd.tyStringStat.sValue		:= p_sAWPushOrPullerAxisErrTxt;
	ELSE
		IF NOT (p_bAWPushOrPullerJogging AND p_eAWPushOrPullerStat = AWActIdle) THEN
	 			tyP0937AWPushOrPuller.tyMotionStd.tyStringStat.sValue		:= p_sAWPushOrPullerStatTxt;
		END_IF

	END_IF

END_ACTION
```

#### Act_OptP0937Mask.st
```iecst
ACTION Act_OptP0937Mask:

	// Interlock Power
	IF p_bAWPushOrPullerAxisErr = TRUE AND p_bAWPushOrPullerPwrOn = FALSE THEN
		fUIInRtStatOff(ADR(tyP0937AWPushOrPuller.tyMotionStd.tyBtnPwr.uiMaskRtStat));
		tyP0937AWPushOrPuller.tyMotionStd.tyBtnPwr.bValue		:= FALSE;
	ELSE
		fUIInRtStatHide(ADR(tyP0937AWPushOrPuller.tyMotionStd.tyBtnPwr.uiMaskRtStat));
	END_IF

	// Interlock Others Move
	IF p_bAWPushOrPullerAxisErr = TRUE OR p_bAWPushOrPullerPwrOn = FALSE THEN
		fUIInRtStatOff(ADR(tyP0937AWPushOrPuller.tyMotionStd.tyBtnOrigin.uiMaskRtStat));
		fUIInRtStatOff(ADR(tyP0937AWPushOrPuller.tyMotionStd.tyBtnMovRel.uiMaskRtStat));
		fUIInRtStatOff(ADR(tyP0937AWPushOrPuller.tyMotionStd.tyBtnJogOpen.uiMaskRtStat));
		fUIInRtStatOff(ADR(tyP0937AWPushOrPuller.tyMotionStd.tyBtnJogClose.uiMaskRtStat));
	ELSE
		fUIInRtStatHide(ADR(tyP0937AWPushOrPuller.tyMotionStd.tyBtnOrigin.uiMaskRtStat));
		fUIInRtStatHide(ADR(tyP0937AWPushOrPuller.tyMotionStd.tyBtnMovRel.uiMaskRtStat));
		fUIInRtStatHide(ADR(tyP0937AWPushOrPuller.tyMotionStd.tyBtnJogOpen.uiMaskRtStat));
		fUIInRtStatHide(ADR(tyP0937AWPushOrPuller.tyMotionStd.tyBtnJogClose.uiMaskRtStat));
	END_IF

	// Interlock Move Absolute
	IF p_bAWPushOrPullerAxisErr = TRUE OR p_bAWPushOrPullerPwrOn = FALSE OR p_bAWPushOrPullerIsHomed = FALSE THEN
		fUIInRtStatOff(ADR(tyP0937AWPushOrPuller.tyAW.tyBtnGo.uiMaskRtStat));
		fUIInRtStatOff(ADR(tyP0937AWPushOrPuller.tyMotionStd.tyBtnMovAbs.uiMaskRtStat));
	ELSE
		fUIInRtStatHide(ADR(tyP0937AWPushOrPuller.tyAW.tyBtnGo.uiMaskRtStat));
		fUIInRtStatHide(ADR(tyP0937AWPushOrPuller.tyMotionStd.tyBtnMovAbs.uiMaskRtStat));
	END_IF

	//Interlock Limit Sensor
	IF tyP0937AWPushOrPuller.tyMotionStd.tyBtnOpenLmtSen.bValue = TRUE THEN
		fUIInRtStatOff(ADR(tyP0937AWPushOrPuller.tyMotionStd.tyBtnJogOpen.uiMaskRtStat));
	END_IF

	IF tyP0937AWPushOrPuller.tyMotionStd.tyBtnCloseLmtSen.bValue = TRUE THEN
		fUIInRtStatOff(ADR(tyP0937AWPushOrPuller.tyMotionStd.tyBtnJogClose.uiMaskRtStat));
	END_IF

	// Interlock When Moving
	IF tyP0937AWPushOrPuller.tyMotionStd.tyBtnOrigin.bRtCompl = TRUE THEN
		fUIInRtStatOff(ADR(tyP0937AWPushOrPuller.tyMotionStd.tyBtnMovAbs.uiMaskRtStat));
		fUIInRtStatOff(ADR(tyP0937AWPushOrPuller.tyMotionStd.tyBtnMovRel.uiMaskRtStat));
		fUIInRtStatOff(ADR(tyP0937AWPushOrPuller.tyMotionStd.tyBtnJogOpen.uiMaskRtStat));
		fUIInRtStatOff(ADR(tyP0937AWPushOrPuller.tyMotionStd.tyBtnJogClose.uiMaskRtStat));
		fUIInRtStatOff(ADR(tyP0937AWPushOrPuller.tyAW.tyBtnGo.uiMaskRtStat));

	ELSIF tyP0937AWPushOrPuller.tyMotionStd.tyBtnMovAbs.bRtCompl = TRUE THEN
		fUIInRtStatOff(ADR(tyP0937AWPushOrPuller.tyMotionStd.tyBtnOrigin.uiMaskRtStat));
		fUIInRtStatOff(ADR(tyP0937AWPushOrPuller.tyMotionStd.tyBtnMovRel.uiMaskRtStat));
		fUIInRtStatOff(ADR(tyP0937AWPushOrPuller.tyMotionStd.tyBtnJogOpen.uiMaskRtStat));
		fUIInRtStatOff(ADR(tyP0937AWPushOrPuller.tyMotionStd.tyBtnJogClose.uiMaskRtStat));
		fUIInRtStatOff(ADR(tyP0937AWPushOrPuller.tyAW.tyBtnGo.uiMaskRtStat));

	ELSIF tyP0937AWPushOrPuller.tyMotionStd.tyBtnMovRel.bRtCompl = TRUE THEN
		fUIInRtStatOff(ADR(tyP0937AWPushOrPuller.tyMotionStd.tyBtnOrigin.uiMaskRtStat));
		fUIInRtStatOff(ADR(tyP0937AWPushOrPuller.tyMotionStd.tyBtnMovAbs.uiMaskRtStat));
		fUIInRtStatOff(ADR(tyP0937AWPushOrPuller.tyMotionStd.tyBtnJogOpen.uiMaskRtStat));
		fUIInRtStatOff(ADR(tyP0937AWPushOrPuller.tyMotionStd.tyBtnJogClose.uiMaskRtStat));
		fUIInRtStatOff(ADR(tyP0937AWPushOrPuller.tyAW.tyBtnGo.uiMaskRtStat));

	ELSIF tyP0937AWPushOrPuller.tyMotionStd.tyBtnJogOpen.bRtCompl = TRUE OR tyP0934AW.tyMotionStd.tyBtnJogOpen.bValue = TRUE THEN
		fUIInRtStatOff(ADR(tyP0937AWPushOrPuller.tyMotionStd.tyBtnOrigin.uiMaskRtStat));
		fUIInRtStatOff(ADR(tyP0937AWPushOrPuller.tyMotionStd.tyBtnMovAbs.uiMaskRtStat));
		fUIInRtStatOff(ADR(tyP0937AWPushOrPuller.tyMotionStd.tyBtnMovRel.uiMaskRtStat));
		fUIInRtStatOff(ADR(tyP0937AWPushOrPuller.tyMotionStd.tyBtnJogClose.uiMaskRtStat));
		fUIInRtStatOff(ADR(tyP0937AWPushOrPuller.tyAW.tyBtnGo.uiMaskRtStat));

	ELSIF tyP0937AWPushOrPuller.tyMotionStd.tyBtnJogClose.bRtCompl = TRUE OR tyP0934AW.tyMotionStd.tyBtnJogClose.bValue = TRUE THEN
		fUIInRtStatOff(ADR(tyP0937AWPushOrPuller.tyMotionStd.tyBtnOrigin.uiMaskRtStat));
		fUIInRtStatOff(ADR(tyP0937AWPushOrPuller.tyMotionStd.tyBtnMovAbs.uiMaskRtStat));
		fUIInRtStatOff(ADR(tyP0937AWPushOrPuller.tyMotionStd.tyBtnMovRel.uiMaskRtStat));
		fUIInRtStatOff(ADR(tyP0937AWPushOrPuller.tyMotionStd.tyBtnJogOpen.uiMaskRtStat));
		fUIInRtStatOff(ADR(tyP0937AWPushOrPuller.tyAW.tyBtnGo.uiMaskRtStat));

	ELSIF tyP0937AWPushOrPuller.tyAW.tyBtnGo.bRtCompl = TRUE THEN
		fUIInRtStatOff(ADR(tyP0937AWPushOrPuller.tyMotionStd.tyBtnOrigin.uiMaskRtStat));
		fUIInRtStatOff(ADR(tyP0937AWPushOrPuller.tyMotionStd.tyBtnMovAbs.uiMaskRtStat));
		fUIInRtStatOff(ADR(tyP0937AWPushOrPuller.tyMotionStd.tyBtnMovRel.uiMaskRtStat));
		fUIInRtStatOff(ADR(tyP0937AWPushOrPuller.tyMotionStd.tyBtnJogOpen.uiMaskRtStat));
		fUIInRtStatOff(ADR(tyP0937AWPushOrPuller.tyMotionStd.tyBtnJogClose.uiMaskRtStat));

	END_IF

	//Axis Error
	IF tyP0937AWPushOrPuller.tyMotionStd.tyBtnPwr.bRtCompl = TRUE THEN
		fUIInRtStatOff(ADR(tyP0937AWPushOrPuller.tyMotionStd.tyBtnRst.uiMaskRtStat));
	ELSE
		fUIInRtStatHide(ADR(tyP0937AWPushOrPuller.tyMotionStd.tyBtnRst.uiMaskRtStat));
	END_IF

END_ACTION
```

#### Act_OptP0937UpdtDat.st
```iecst
ACTION Act_OptP0937UpdtDat:

	tyP0937AWPushOrPuller.tyMotionStd.tyNumCurrPos.diValue		:= p_diAWPushOrPullerActualPos;
	tyP0937AWPushOrPuller.tyMotionStd.tyNumErrCode.diValue		:= UDINT_TO_DINT(p_udiAWPushOrPullerAxisErrID);
	tyP0937AWPushOrPuller.tyMotionStd.tyBitmapPwr.usiValueIdx		:= BOOL_TO_USINT(p_bAWPushOrPullerPwrOn);
	tyP0937AWPushOrPuller.tyMotionStd.tyBitmapRst.usiValueIdx		:= BOOL_TO_USINT(NOT p_bAWPushOrPullerAxisErr);
	tyP0937AWPushOrPuller.tyMotionStd.tyBitmapOrigin.usiValueIdx	:= BOOL_TO_USINT(p_bAWPushOrPullerIsHomed);
	tyP0937AWPushOrPuller.tyMotionStd.tyBtnOpenLmtSen.bValue		:= p_bAWPushOrPullerCloseSen;
	tyP0937AWPushOrPuller.tyMotionStd.tyBtnCloseLmtSen.bValue		:= p_bAWPushOrPullerOpenSen;

	IF p_bAWPushOrPullerIsHomed = TRUE THEN
		IF p_diAWPushOrPullerActualPos <= (p_tyNtParamCurr.tyProdRcpWidth.diMax / 2) THEN
			tyP0937AWPushOrPuller.tyMotionStd.tyBitmapMc.uiValueIdx 	:= 38;
		ELSE
			tyP0937AWPushOrPuller.tyMotionStd.tyBitmapMc.uiValueIdx 	:= 39;
		END_IF
	ELSE
		tyP0937AWPushOrPuller.tyMotionStd.tyBitmapMc.uiValueIdx	:= 38;
	END_IF

	IF p_tyNtParamCurr.eProjMag = ULMagTriple AND p_tyNtParamCurr.bMagAutoVerifyPrep = FALSE AND p_tyNtParamCurr.bProjMotorizedPusherPrep = TRUE THEN
	IF 	tyP0937AWPushOrPuller.tyMotionStd.tyBitmapMc.uiValueIdx < 400 THEN
		tyP0937AWPushOrPuller.tyMotionStd.tyBitmapMc.uiValueIdx	:= tyP0937AWPushOrPuller.tyMotionStd.tyBitmapMc.uiValueIdx + 400;
	END_IF
	END_IF
END_ACTION
```

#### Act_OptP0937Keypad.st
```iecst
ACTION Act_OptP0937Keypad:

	IF fUIOutRtStatTPIsOpen(ADR(tyP0937AWPushOrPuller.tyAW.tyNumNewWidth.uiRtStat)) = TRUE THEN
		tyProperty.tyKeypad.tyStringTitle.sKeypadTitle		:= tyP0937AWPushOrPuller.tyAW.tyNumNewWidth.sKeypadTitle;

	ELSIF fUIOutRtStatTPIsOpen(ADR(tyP0937AWPushOrPuller.tyMotionStd.tyNumTargetPos.uiRtStat)) = TRUE THEN
		tyProperty.tyKeypad.tyStringTitle.sKeypadTitle		:= tyP0937AWPushOrPuller.tyMotionStd.tyNumTargetPos.sKeypadTitle;

	ELSIF fUIOutRtStatTPIsOpen(ADR(tyP0937AWPushOrPuller.tyMotionStd.tyNumStepSize.uiRtStat)) = TRUE THEN
		tyProperty.tyKeypad.tyStringTitle.sKeypadTitle		:= tyP0937AWPushOrPuller.tyMotionStd.tyNumStepSize.sKeypadTitle;

	ELSIF fUIOutRtStatTPIsOpen(ADR(tyP0937AWPushOrPuller.tyMotionStd.tyNumNomSpd.uiRtStat)) = TRUE THEN
		tyProperty.tyKeypad.tyStringTitle.sKeypadTitle		:= tyP0937AWPushOrPuller.tyMotionStd.tyNumNomSpd.sKeypadTitle;

	ELSIF fUIOutRtStatTPIsOpen(ADR(tyP0937AWPushOrPuller.tyMotionStd.tyNumSlwSpd.uiRtStat)) = TRUE THEN
		tyProperty.tyKeypad.tyStringTitle.sKeypadTitle		:= tyP0937AWPushOrPuller.tyMotionStd.tyNumSlwSpd.sKeypadTitle;

	END_IF

END_ACTION
```

#### Act_OptP0937RstMnl.st
```iecst
ACTION Act_OptP0937RstMnl:

	IF EDGEPOS((bManualMod = FALSE) OR (p_eAWPushOrPullerStatus = Error)) THEN

		eAWPushOrPullerAct	:= AWActIdle;

		bJogSlow				:= FALSE;
		bJogFast				:= FALSE;
		fbJogSlowToFastDlyTm.IN	:= FALSE;

		tyP0937AWPushOrPuller.tyAW.tyBtnGo.bRtCompl					:= FALSE;
		tyP0937AWPushOrPuller.tyAW.tyBtnGo.bValue					:= FALSE;
		tyP0937AWPushOrPuller.tyAW.tyBtnGo.bRtLk					:= FALSE;
		tyP0937AWPushOrPuller.tyAW.tyBtnGo.uiMaskRtStat.0			:= FALSE;

		tyP0937AWPushOrPuller.tyMotionStd.tyBtnPwr.bRtCompl			:= FALSE;
		tyP0937AWPushOrPuller.tyMotionStd.tyBtnStop.bRtCompl		:= FALSE;
		tyP0937AWPushOrPuller.tyMotionStd.tyBtnOrigin.bRtCompl		:= FALSE;
		tyP0937AWPushOrPuller.tyMotionStd.tyBtnRst.bRtCompl			:= FALSE;
		tyP0937AWPushOrPuller.tyMotionStd.tyBtnMovAbs.bRtCompl		:= FALSE;
		tyP0937AWPushOrPuller.tyMotionStd.tyBtnMovRel.bRtCompl		:= FALSE;
		tyP0937AWPushOrPuller.tyMotionStd.tyBtnJogOpen.bRtCompl		:= FALSE;
		tyP0937AWPushOrPuller.tyMotionStd.tyBtnJogClose.bRtCompl	:= FALSE;

		tyP0937AWPushOrPuller.tyMotionStd.tyBtnPwr.bValue			:= FALSE;
		tyP0937AWPushOrPuller.tyMotionStd.tyBtnStop.bValue			:= TRUE;
		tyP0937AWPushOrPuller.tyMotionStd.tyBtnOrigin.bValue		:= FALSE;
		tyP0937AWPushOrPuller.tyMotionStd.tyBtnRst.bValue			:= FALSE;
		tyP0937AWPushOrPuller.tyMotionStd.tyBtnMovAbs.bValue		:= FALSE;
		tyP0937AWPushOrPuller.tyMotionStd.tyBtnMovRel.bValue		:= FALSE;
		tyP0937AWPushOrPuller.tyMotionStd.tyBtnJogOpen.bValue		:= FALSE;
		tyP0937AWPushOrPuller.tyMotionStd.tyBtnJogClose.bValue		:= FALSE;

		tyP0937AWPushOrPuller.tyMotionStd.tyBtnPwr.bRtLk			:= FALSE;
		tyP0937AWPushOrPuller.tyMotionStd.tyBtnStop.bRtLk			:= TRUE;
		tyP0937AWPushOrPuller.tyMotionStd.tyBtnOrigin.bRtLk			:= FALSE;
		tyP0937AWPushOrPuller.tyMotionStd.tyBtnRst.bRtLk			:= FALSE;
		tyP0937AWPushOrPuller.tyMotionStd.tyBtnMovAbs.bRtLk			:= FALSE;
		tyP0937AWPushOrPuller.tyMotionStd.tyBtnMovRel.bRtLk			:= FALSE;
		tyP0937AWPushOrPuller.tyMotionStd.tyBtnJogOpen.bRtLk		:= FALSE;
		tyP0937AWPushOrPuller.tyMotionStd.tyBtnJogClose.bRtLk		:= FALSE;

		tyP0937AWPushOrPuller.tyMotionStd.tyBtnPwr.uiMaskRtStat		:= TRUE;
		tyP0937AWPushOrPuller.tyMotionStd.tyBtnOrigin.uiMaskRtStat	:= FALSE;
		tyP0937AWPushOrPuller.tyMotionStd.tyBtnRst.uiMaskRtStat		:= TRUE;
		tyP0937AWPushOrPuller.tyMotionStd.tyBtnMovAbs.uiMaskRtStat	:= FALSE;
		tyP0937AWPushOrPuller.tyMotionStd.tyBtnMovRel.uiMaskRtStat	:= FALSE;
		tyP0937AWPushOrPuller.tyMotionStd.tyBtnJogOpen.uiMaskRtStat	:= FALSE;
		tyP0937AWPushOrPuller.tyMotionStd.tyBtnJogClose.uiMaskRtStat	:= FALSE;

	END_IF

END_ACTION
```

#### Act_EntP0938Disp.st
```iecst
ACTION Act_EntP0938Disp:

	CASE p_tyMagRcpCurrRcp.usiMagModel OF
		0://CAB706.2
			bSmallMagLimSen1:= TRUE;
			bSmallMagLimSen2:= TRUE;
			bSmallMagLimSen3:= TRUE;
			bSmallMagLimSen4:= TRUE;
		1://CAB716.2
			bSmallMagLimSen1:= TRUE;
			bSmallMagLimSen2:= TRUE;
			bSmallMagLimSen3:= TRUE;
			bSmallMagLimSen4:= TRUE;
		2://CAB717.2
			bSmallMagLimSen1:= FALSE;
			bSmallMagLimSen2:= FALSE;
			bSmallMagLimSen3:= FALSE;
			bSmallMagLimSen4:= FALSE;
	END_CASE

	//Access Address
	IF bDispMagAW1 = TRUE THEN

		(*Magazine Auto Width 1*)
		p_tyC0001MotionStd ACCESS ADR(tyP0938MagAW.tyMotionStd1);

		p_tyC0002FullMask ACCESS ADR(tyP0938MagAW.tyFullMaskHide);

		IF p_tyNtParamCurr.eProjMag = ULMagDual THEN
			p_tyC0004Navi ACCESS ADR(tyP0938MagAW.tyNavi2Lyr1);
		ELSE
			p_tyC0004Navi ACCESS ADR(tyP0938MagAW.tyNavi3Lyr1);
		END_IF

		p_tyC0005Main ACCESS ADR(tyCommon.tyMain);

		p_tyC0007Notif ACCESS ADR(tyCommon.tyNotif);

		p_tyC0008MsgBox ACCESS ADR(tyP0938MagAW.tyMsgBoxHide);

		p_tyC0009Info ACCESS ADR(tyCommon.tyInfo);

		p_tyP0938MagAW ACCESS ADR(tyP0938MagAW.tyMagAW1);

	ELSIF bDispMagAW2 = TRUE THEN

		(*Magazine Auto Width 2*)
		p_tyC0001MotionStd ACCESS ADR(tyP0938MagAW.tyMotionStd2);

		p_tyC0002FullMask ACCESS ADR(tyP0938MagAW.tyFullMaskHide);

		IF p_tyNtParamCurr.eProjMag = ULMagDual THEN
			p_tyC0004Navi ACCESS ADR(tyP0938MagAW.tyNavi2Lyr2);
		ELSE
			p_tyC0004Navi ACCESS ADR(tyP0938MagAW.tyNavi3Lyr2);
		END_IF

		p_tyC0005Main ACCESS ADR(tyCommon.tyMain);

		p_tyC0007Notif ACCESS ADR(tyCommon.tyNotif);

		p_tyC0008MsgBox ACCESS ADR(tyP0938MagAW.tyMsgBoxHide);

		p_tyC0009Info ACCESS ADR(tyCommon.tyInfo);

		p_tyP0938MagAW ACCESS ADR(tyP0938MagAW.tyMagAW2);

	ELSIF bDispMagAW3 = TRUE THEN

		(*Magazine Auto Width 3*)
		p_tyC0001MotionStd ACCESS ADR(tyP0938MagAW.tyMotionStd3);

		p_tyC0002FullMask ACCESS ADR(tyP0938MagAW.tyFullMaskHide);

		p_tyC0004Navi ACCESS ADR(tyP0938MagAW.tyNavi3Lyr3);

		p_tyC0005Main ACCESS ADR(tyCommon.tyMain);

		p_tyC0007Notif ACCESS ADR(tyCommon.tyNotif);

		p_tyC0008MsgBox ACCESS ADR(tyP0938MagAW.tyMsgBoxHide);

		p_tyC0009Info ACCESS ADR(tyCommon.tyInfo);

		p_tyP0938MagAW ACCESS ADR(tyP0938MagAW.tyMagAW3);

	END_IF

	//Display
	(*Magazine Auto Width 1*)
	tyP0938MagAW.tyMagAW1.tyNumNewWidth.diValue	:= p_tyProdRcpCurrRcp0.diWidthInUM;
	tyP0938MagAW.tyMagAW1.tyBtnEngage.bValue	:= p_bMag1AWEngageExtCtrl;
	tyP0938MagAW.tyMagAW1.tyBtnDisengage.bValue	:= p_bMag1AWEngageRetCtrl;

	tyP0938MagAW.tyMotionStd1.tyBtnPwr.bValue	:= p_bMagAWOpen1PwrOn;

	(*Magazine Auto Width 2*)
	tyP0938MagAW.tyMagAW2.tyNumNewWidth.diValue	:= p_tyProdRcpCurrRcp0.diWidthInUM;
	tyP0938MagAW.tyMagAW2.tyBtnEngage.bValue	:= p_bMag2AWEngageExtCtrl;
	tyP0938MagAW.tyMagAW2.tyBtnDisengage.bValue	:= p_bMag2AWEngageRetCtrl;

	tyP0938MagAW.tyMotionStd2.tyBtnPwr.bValue	:= p_bMagAWOpen2PwrOn;

	(*Magazine Auto Width 3*)
	tyP0938MagAW.tyMagAW3.tyNumNewWidth.diValue	:= p_tyProdRcpCurrRcp0.diWidthInUM;
	tyP0938MagAW.tyMagAW3.tyBtnEngage.bValue	:= p_bMag3AWEngageExtCtrl;
	tyP0938MagAW.tyMagAW3.tyBtnDisengage.bValue	:= p_bMag3AWEngageRetCtrl;

	tyP0938MagAW.tyMotionStd3.tyBtnPwr.bValue	:= p_bMagAWOpen3PwrOn;

END_ACTION
```

#### Act_OptP0938Navi.st
```iecst
ACTION Act_OptP0938Navi:

	CASE p_tyNtParamCurr.eProjMag OF
		ULMagDual:
			IF tyP0938MagAW.tyNavi2Lyr1.tyBtnBack.bRtCompl = TRUE OR tyP0938MagAW.tyNavi2Lyr2.tyBtnBack.bRtCompl = TRUE THEN
				tyP0938MagAW.tyNavi2Lyr1.tyBtnBack.bRtCompl := FALSE;
				tyP0938MagAW.tyNavi2Lyr1.tyBtnBack.bValue	:= FALSE;
				tyP0938MagAW.tyNavi2Lyr2.tyBtnBack.bRtCompl := FALSE;
				tyP0938MagAW.tyNavi2Lyr2.tyBtnBack.bValue	:= FALSE;

				eChgPage	:= UIP0920MtrNPneuCtrl;

			ELSIF tyP0938MagAW.tyNavi2Lyr1.tyBtnLeft.bRtCompl = TRUE OR tyP0938MagAW.tyNavi2Lyr1.tyBtnRgt.bRtCompl = TRUE THEN
				tyP0938MagAW.tyNavi2Lyr1.tyBtnLeft.bRtCompl	:= FALSE;
				tyP0938MagAW.tyNavi2Lyr1.tyBtnRgt.bRtCompl	:= FALSE;

				bDispMagAW1	:= FALSE;
				bDispMagAW2	:= TRUE;
				bDispMagAW3	:= FALSE;

				p_tyC0004Navi ACCESS ADR(tyP0938MagAW.tyNavi2Lyr2);

				p_tyC0001MotionStd ACCESS ADR(tyP0938MagAW.tyMotionStd2);

				p_tyP0938MagAW ACCESS ADR(tyP0938MagAW.tyMagAW2);

			ELSIF tyP0938MagAW.tyNavi2Lyr2.tyBtnLeft.bRtCompl = TRUE OR tyP0938MagAW.tyNavi2Lyr2.tyBtnRgt.bRtCompl = TRUE THEN
				tyP0938MagAW.tyNavi2Lyr2.tyBtnLeft.bRtCompl	:= FALSE;
				tyP0938MagAW.tyNavi2Lyr2.tyBtnRgt.bRtCompl	:= FALSE;

				bDispMagAW1	:= TRUE;
				bDispMagAW2	:= FALSE;
				bDispMagAW3	:= FALSE;

				p_tyC0004Navi ACCESS ADR(tyP0938MagAW.tyNavi2Lyr1);

				p_tyC0001MotionStd ACCESS ADR(tyP0938MagAW.tyMotionStd1);

				p_tyP0938MagAW ACCESS ADR(tyP0938MagAW.tyMagAW1);

			END_IF

		ULMagTriple:
			IF tyP0938MagAW.tyNavi3Lyr1.tyBtnBack.bRtCompl = TRUE OR tyP0938MagAW.tyNavi3Lyr2.tyBtnBack.bRtCompl = TRUE OR tyP0938MagAW.tyNavi3Lyr3.tyBtnBack.bRtCompl = TRUE THEN
				tyP0938MagAW.tyNavi3Lyr1.tyBtnBack.bRtCompl := FALSE;
				tyP0938MagAW.tyNavi3Lyr1.tyBtnBack.bValue	:= FALSE;
				tyP0938MagAW.tyNavi3Lyr2.tyBtnBack.bRtCompl := FALSE;
				tyP0938MagAW.tyNavi3Lyr2.tyBtnBack.bValue	:= FALSE;
				tyP0938MagAW.tyNavi3Lyr3.tyBtnBack.bRtCompl := FALSE;
				tyP0938MagAW.tyNavi3Lyr3.tyBtnBack.bValue	:= FALSE;

				eChgPage	:= UIP0920MtrNPneuCtrl;

			ELSIF tyP0938MagAW.tyNavi3Lyr1.tyBtnLeft.bRtCompl = TRUE THEN
				tyP0938MagAW.tyNavi3Lyr1.tyBtnLeft.bRtCompl	:= FALSE;

				bDispMagAW1	:= FALSE;
				bDispMagAW2	:= FALSE;
				bDispMagAW3	:= TRUE;

				p_tyC0004Navi ACCESS ADR(tyP0938MagAW.tyNavi3Lyr3);

				p_tyC0001MotionStd ACCESS ADR(tyP0938MagAW.tyMotionStd3);

				p_tyP0938MagAW ACCESS ADR(tyP0938MagAW.tyMagAW3);

			ELSIF tyP0938MagAW.tyNavi3Lyr1.tyBtnRgt.bRtCompl = TRUE THEN
				tyP0938MagAW.tyNavi3Lyr1.tyBtnRgt.bRtCompl	:= FALSE;

				bDispMagAW1	:= FALSE;
				bDispMagAW2	:= TRUE;
				bDispMagAW3	:= FALSE;

				p_tyC0004Navi ACCESS ADR(tyP0938MagAW.tyNavi3Lyr2);

				p_tyC0001MotionStd ACCESS ADR(tyP0938MagAW.tyMotionStd2);

				p_tyP0938MagAW ACCESS ADR(tyP0938MagAW.tyMagAW2);

			ELSIF tyP0938MagAW.tyNavi3Lyr2.tyBtnLeft.bRtCompl = TRUE THEN
				tyP0938MagAW.tyNavi3Lyr2.tyBtnLeft.bRtCompl	:= FALSE;

				bDispMagAW1	:= TRUE;
				bDispMagAW2	:= FALSE;
				bDispMagAW3	:= FALSE;

				p_tyC0004Navi ACCESS ADR(tyP0938MagAW.tyNavi3Lyr1);

				p_tyC0001MotionStd ACCESS ADR(tyP0938MagAW.tyMotionStd1);

				p_tyP0938MagAW ACCESS ADR(tyP0938MagAW.tyMagAW1);

			ELSIF tyP0938MagAW.tyNavi3Lyr2.tyBtnRgt.bRtCompl = TRUE THEN
				tyP0938MagAW.tyNavi3Lyr2.tyBtnRgt.bRtCompl	:= FALSE;

				bDispMagAW1	:= FALSE;
				bDispMagAW2	:= FALSE;
				bDispMagAW3	:= TRUE;

				p_tyC0004Navi ACCESS ADR(tyP0938MagAW.tyNavi3Lyr3);

				p_tyC0001MotionStd ACCESS ADR(tyP0938MagAW.tyMotionStd3);

				p_tyP0938MagAW ACCESS ADR(tyP0938MagAW.tyMagAW3);

			ELSIF tyP0938MagAW.tyNavi3Lyr3.tyBtnLeft.bRtCompl = TRUE THEN
				tyP0938MagAW.tyNavi3Lyr3.tyBtnLeft.bRtCompl	:= FALSE;

				bDispMagAW1	:= FALSE;
				bDispMagAW2	:= TRUE;
				bDispMagAW3	:= FALSE;

				p_tyC0004Navi ACCESS ADR(tyP0938MagAW.tyNavi3Lyr2);

				p_tyC0001MotionStd ACCESS ADR(tyP0938MagAW.tyMotionStd2);

				p_tyP0938MagAW ACCESS ADR(tyP0938MagAW.tyMagAW2);

			ELSIF tyP0938MagAW.tyNavi3Lyr3.tyBtnRgt.bRtCompl = TRUE THEN
				tyP0938MagAW.tyNavi3Lyr3.tyBtnRgt.bRtCompl	:= FALSE;

				bDispMagAW1	:= TRUE;
				bDispMagAW2	:= FALSE;
				bDispMagAW3	:= FALSE;

				p_tyC0004Navi ACCESS ADR(tyP0938MagAW.tyNavi3Lyr1);

				p_tyC0001MotionStd ACCESS ADR(tyP0938MagAW.tyMotionStd1);

				p_tyP0938MagAW ACCESS ADR(tyP0938MagAW.tyMagAW1);

			END_IF

	END_CASE

END_ACTION
```

#### Act_OptP0938FullMask.st
```iecst
ACTION Act_OptP0938FullMask:

	IF eCurrPage = UIP0938MagAW THEN

		IF p_tyDI.bEStopSig = FALSE THEN
			p_tyC0002FullMask ACCESS ADR(tyP0938MagAW.tyFullMaskEStop);

		ELSIF p_tyDI.bCoverSWSig = FALSE THEN
			p_tyC0002FullMask ACCESS ADR(tyP0938MagAW.tyFullMaskCWSig);

		ELSIF p_tyDI.bSafetyRlySig = FALSE THEN
			p_tyC0002FullMask ACCESS ADR(tyP0938MagAW.tyFullMaskSafetyRly);

		ELSIF bDispMagAW1 AND p_tyBuffer1BffrStat.bBffrMty = FALSE AND p_tyDI.bMagPresentSen1  THEN
			p_tyC0002FullMask ACCESS ADR(tyP0938MagAW.tyFullMaskMag1NotMty);

		ELSIF bDispMagAW2 AND p_tyBuffer2BffrStat.bBffrMty = FALSE AND p_tyDI.bMagPresentSen2 THEN
			p_tyC0002FullMask ACCESS ADR(tyP0938MagAW.tyFullMaskMag2NotMty);

		ELSIF bDispMagAW3 AND p_tyBuffer3BffrStat.bBffrMty = FALSE AND p_tyDI.bMagPresentSen3 THEN
			p_tyC0002FullMask ACCESS ADR(tyP0938MagAW.tyFullMaskMag3NotMty);

		ELSE
			p_tyC0002FullMask ACCESS ADR(tyP0938MagAW.tyFullMaskHide);

		END_IF

	END_IF

END_ACTION
```
